C01819=1024.625,112.284,392.531,168.036,48.141,158.964
C01820=1024.630,112.533,392.511,168.039,48.136,158.963
C01821=1024.636,112.782,392.492,168.042,48.132,158.963
C01822=1024.642,113.032,392.473,168.044,48.128,158.962
C01823=1024.648,113.281,392.453,168.047,48.124,158.962
C01824=1024.654,113.530,392.434,168.049,48.119,158.962
C01825=1024.659,113.780,392.414,168.052,48.115,158.961
C01826=1024.665,114.028,392.395,168.055,48.111,158.961
C01827=1024.670,114.277,392.376,168.057,48.107,158.960
C01828=1024.676,114.527,392.356,168.060,48.103,158.960
C01829=1024.681,114.776,392.336,168.063,48.099,158.959
C01830=1024.687,115.025,392.317,168.065,48.094,158.959
C01831=1024.693,115.274,392.297,168.069,48.090,158.959
C01832=1024.699,115.523,392.277,168.072,48.086,158.958
C01833=1024.704,115.773,392.258,168.074,48.082,158.958
C01834=1024.710,116.022,392.238,168.077,48.077,158.957
C01835=1024.716,116.271,392.219,168.080,48.073,158.957
C01836=1024.722,116.520,392.199,168.082,48.069,158.956
C01837=1024.727,116.770,392.179,168.085,48.065,158.956
C01838=1024.733,117.018,392.159,168.087,48.061,158.955
C01839=1024.738,117.267,392.140,168.090,48.057,158.955
C01840=1024.744,117.517,392.121,168.094,48.052,158.955
C01841=1024.750,117.765,392.101,168.097,48.048,158.954
C01842=1024.755,118.015,392.082,168.099,48.044,158.954
C01843=1024.761,118.264,392.062,168.102,48.040,158.953
C01844=1024.766,118.513,392.042,168.104,48.035,158.953
C01845=1024.772,118.762,392.022,168.107,48.031,158.952
C01846=1024.778,119.012,392.003,168.110,48.027,158.952
C01847=1024.784,119.260,391.983,168.112,48.022,158.951
C01848=1024.790,119.510,391.964,168.116,48.018,158.951
C01849=1024.796,119.759,391.944,168.118,48.014,158.950
C01850=1024.801,120.008,391.924,168.121,48.010,158.950
C01851=1024.807,120.257,391.904,168.124,48.005,158.950
C01852=1024.812,120.507,391.885,168.127,48.002,158.949
C01853=1024.818,120.755,391.865,168.129,47.997,158.949
C01854=1024.824,121.005,391.845,168.132,47.993,158.948
C01855=1024.830,121.254,391.826,168.135,47.988,158.948
C01856=1024.836,121.502,391.806,168.138,47.984,158.947
C01857=1024.842,121.752,391.786,168.141,47.980,158.947
C01858=1024.847,122.001,391.766,168.143,47.976,158.946
C01859=1024.853,122.250,391.747,168.146,47.972,158.946
C01860=1024.859,122.500,391.726,168.149,47.967,158.946
C01861=1024.865,122.749,391.706,168.152,47.963,158.945
C01862=1024.871,122.998,391.687,168.155,47.959,158.945
C01863=1024.877,123.247,391.667,168.157,47.954,158.944
C01864=1024.883,123.531,391.644,168.161,47.949,158.944
C01865=1024.890,123.815,391.621,168.164,47.945,158.943
C01866=1024.896,124.099,391.599,168.167,47.940,158.943
C01867=1024.903,124.383,391.577,168.170,47.935,158.942
C01868=1024.909,124.632,391.558,168.173,47.931,158.942
C01869=1024.914,124.882,391.537,168.176,47.926,158.941
C01870=1024.920,125.131,391.517,168.179,47.922,158.941
C01871=1024.926,125.380,391.497,168.182,47.918,158.940
C01872=1024.932,125.629,391.477,168.184,47.913,158.940
C01873=1024.938,125.878,391.457,168.187,47.909,158.939
C01874=1024.944,126.127,391.438,168.191,47.905,158.939
C01875=1024.949,126.376,391.418,168.193,47.901,158.938
C01876=1024.955,126.625,391.398,168.196,47.896,158.938
C01877=1024.961,126.874,391.378,168.198,47.892,158.937
C01878=1024.967,127.124,391.358,168.202,47.888,158.937
C01879=1024.973,127.373,391.338,168.205,47.883,158.937
C01880=1024.979,127.622,391.318,168.207,47.879,158.936
C01881=1024.984,127.872,391.298,168.210,47.875,158.936
C01882=1024.990,128.120,391.278,168.214,47.870,158.935
C01883=1024.996,128.369,391.258,168.216,47.866,158.935
C01884=1025.003,128.619,391.238,168.219,47.862,158.934
C01885=1025.009,128.868,391.219,168.221,47.857,158.934
C01886=1025.015,129.117,391.199,168.225,47.853,158.933
C01887=1025.020,129.366,391.178,168.228,47.849,158.933
C01888=1025.026,129.615,391.158,168.230,47.844,158.932
C01889=1025.032,129.864,391.138,168.233,47.841,158.932
C01890=1025.038,130.114,391.119,168.237,47.836,158.932
C01891=1025.043,130.363,391.098,168.239,47.832,158.931
C01892=1025.049,130.612,391.078,168.242,47.828,158.931
C01893=1025.055,130.861,391.058,168.245,47.824,158.930
C01894=1025.061,131.110,391.038,168.247,47.819,158.930
C01895=1025.066,131.359,391.017,168.251,47.815,158.929
C01896=1025.072,131.608,390.997,168.254,47.811,158.929
C01897=1025.078,131.857,390.976,168.256,47.807,158.928
C01898=1025.084,132.106,390.956,168.259,47.802,158.928
C01899=1025.089,132.355,390.936,168.262,47.799,158.928
C01900=1025.095,132.604,390.916,168.265,47.794,158.927
C01901=1025.101,132.854,390.895,168.268,47.790,158.927
C01902=1025.107,133.103,390.875,168.271,47.786,158.926
C01903=1025.112,133.352,390.855,168.273,47.782,158.926
C01904=1025.118,133.601,390.835,168.276,47.777,158.925
C01905=1025.123,133.850,390.814,168.280,47.773,158.925
C01906=1025.130,134.099,390.794,168.282,47.769,158.924
C01907=1025.135,134.349,390.773,168.285,47.765,158.924
C01908=1025.141,134.597,390.753,168.288,47.761,158.924
C01909=1025.146,134.846,390.733,168.291,47.756,158.923
C01910=1025.153,135.095,390.712,168.294,47.753,158.923
C01911=1025.159,135.344,390.691,168.297,47.748,158.922
C01912=1025.165,135.593,390.671,168.300,47.744,158.922
C01913=1025.170,135.842,390.650,168.303,47.740,158.921
C01914=1025.176,136.092,390.630,168.306,47.736,158.921
C01915=1025.182,136.341,390.610,168.309,47.731,158.921
C01916=1025.187,136.590,390.589,168.311,47.727,158.920
C01917=1025.193,136.839,390.569,168.314,47.723,158.920
C01918=1025.199,137.088,390.547,168.318,47.719,158.919
C01919=1025.205,137.337,390.528,168.320,47.714,158.919
C01920=1025.210,137.586,390.507,168.323,47.711,158.918
C01921=1025.216,137.836,390.486,168.326,47.706,158.918
C01922=1025.222,138.085,390.466,168.329,47.702,158.918
C01923=1025.228,138.333,390.445,168.332,47.698,158.917
C01924=1025.234,138.582,390.425,168.335,47.694,158.917
C01925=1025.240,138.832,390.404,168.338,47.690,158.916
C01926=1025.245,139.081,390.383,168.341,47.685,158.916
C01927=1025.250,139.330,390.362,168.344,47.682,158.915
C01928=1025.257,139.614,390.339,168.348,47.677,158.915
C01929=1025.264,139.898,390.315,168.351,47.672,158.915
C01930=1025.270,140.182,390.291,168.354,47.668,158.914
C01931=1025.277,140.465,390.268,168.357,47.663,158.914
C01932=1025.282,140.714,390.247,168.361,47.658,158.913
C01933=1025.288,140.964,390.226,168.364,47.654,158.913
C01934=1025.294,141.213,390.205,168.366,47.651,158.912
C01935=1025.299,141.462,390.184,168.369,47.646,158.912
C01936=1025.306,141.711,390.164,168.373,47.642,158.911
C01937=1025.311,141.960,390.143,168.375,47.638,158.911
C01938=1025.316,142.209,390.122,168.378,47.634,158.911
C01939=1025.323,142.458,390.101,168.381,47.630,158.910
C01940=1025.329,142.707,390.081,168.384,47.625,158.910
C01941=1025.334,142.956,390.060,168.387,47.622,158.909
C01942=1025.340,143.205,390.039,168.390,47.617,158.909
C01943=1025.345,143.455,390.018,168.393,47.613,158.908
C01944=1025.351,143.703,389.997,168.397,47.609,158.908
C01945=1025.357,143.953,389.976,168.399,47.605,158.908
C01946=1025.363,144.201,389.955,168.402,47.601,158.907
C01947=1025.369,144.451,389.934,168.405,47.596,158.907
C01948=1025.374,144.700,389.914,168.408,47.592,158.906
C01949=1025.380,144.949,389.892,168.411,47.589,158.906
C01950=1025.386,145.198,389.872,168.415,47.584,158.905
C01951=1025.392,145.447,389.851,168.418,47.580,158.905
C01952=1025.398,145.696,389.830,168.420,47.576,158.905
C01953=1025.403,145.945,389.809,168.423,47.572,158.904
C01954=1025.409,146.195,389.788,168.427,47.568,158.904
C01955=1025.415,146.443,389.766,168.429,47.563,158.903
C01956=1025.420,146.692,389.745,168.432,47.560,158.903
C01957=1025.426,146.942,389.724,168.436,47.556,158.903
C01958=1025.432,147.190,389.703,168.439,47.551,158.902
C01959=1025.438,147.440,389.683,168.441,47.547,158.902
C01960=1025.444,147.688,389.661,168.445,47.543,158.901
C01961=1025.450,147.937,389.640,168.448,47.539,158.901
C01962=1025.454,148.187,389.619,168.451,47.535,158.900
C01963=1025.460,148.435,389.597,168.453,47.531,158.900
C01964=1025.466,148.684,389.576,168.457,47.527,158.900
C01965=1025.471,148.934,389.555,168.460,47.523,158.899
C01966=1025.478,149.183,389.533,168.463,47.519,158.899
C01967=1025.483,149.431,389.512,168.466,47.514,158.898
C01968=1025.489,149.681,389.491,168.469,47.511,158.898
C01969=1025.495,149.930,389.470,168.472,47.507,158.898
C01970=1025.501,150.179,389.448,168.476,47.502,158.897
C01971=1025.506,150.428,389.428,168.478,47.498,158.897
C01972=1025.512,150.677,389.406,168.481,47.495,158.896
C01973=1025.518,150.926,389.385,168.485,47.491,158.896
C01974=1025.524,151.175,389.363,168.488,47.486,158.896
C01975=1025.529,151.424,389.343,168.490,47.482,158.895
C01976=1025.535,151.673,389.321,168.494,47.478,158.895
C01977=1025.541,151.922,389.300,168.497,47.474,158.894
C01978=1025.547,152.171,389.278,168.500,47.470,158.894
C01979=1025.553,152.419,389.257,168.504,47.466,158.894
C01980=1025.558,152.669,389.235,168.506,47.462,158.893
C01981=1025.563,152.918,389.214,168.509,47.458,158.893
C01982=1025.569,153.167,389.193,168.513,47.454,158.892
C01983=1025.575,153.416,389.171,168.516,47.450,158.892
C01984=1025.581,153.665,389.150,168.518,47.446,158.892
C01985=1025.587,153.913,389.128,168.522,47.442,158.891
C01986=1025.593,154.163,389.107,168.525,47.438,158.891
C01987=1025.598,154.413,389.085,168.528,47.434,158.890
C01988=1025.604,154.661,389.064,168.531,47.429,158.890
C01989=1025.610,154.910,389.042,168.534,47.426,158.890
C01990=1025.615,155.159,389.021,168.537,47.422,158.889
C01991=1025.621,155.408,388.999,168.541,47.418,158.889
C01992=1025.628,155.692,388.974,168.544,47.413,158.888
C01993=1025.634,155.975,388.950,168.548,47.409,158.888
C01994=1025.640,156.259,388.925,168.552,47.404,158.887
C01995=1025.647,156.542,388.900,168.555,47.399,158.887
C01996=1025.653,156.792,388.879,168.558,47.395,158.887
C01997=1025.659,157.040,388.857,168.561,47.392,158.886
C01998=1025.664,157.290,388.835,168.565,47.388,158.886
C01999=1025.670,157.538,388.814,168.568,47.384,158.886
C02000=1025.676,157.787,388.792,168.570,47.379,158.885
C02001=1025.682,158.037,388.771,168.574,47.375,158.885
C02002=1025.687,158.285,388.749,168.577,47.372,158.884
C02003=1025.693,158.535,388.727,168.581,47.368,158.884
C02004=1025.699,158.783,388.706,168.583,47.363,158.883
C02005=1025.705,159.032,388.684,168.586,47.359,158.883
C02006=1025.711,159.281,388.663,168.590,47.355,158.883
C02007=1025.716,159.530,388.641,168.593,47.352,158.882
C02008=1025.721,159.771,388.619,168.596,47.348,158.882
C02009=1025.727,160.013,388.598,168.599,47.344,158.882
C02010=1025.732,160.254,388.576,168.602,47.340,158.881
C02011=1025.737,160.495,388.555,168.605,47.336,158.881
C02012=1025.743,160.737,388.534,168.608,47.333,158.881
C02013=1025.748,160.978,388.512,168.611,47.330,158.880
C02014=1025.753,161.220,388.491,168.614,47.326,158.880
C02015=1025.758,161.460,388.469,168.618,47.322,158.880
C02016=1025.765,161.709,388.447,168.621,47.318,158.879
C02017=1025.770,161.958,388.425,168.624,47.314,158.879
C02018=1025.775,162.207,388.403,168.628,47.310,158.879
C02019=1025.781,162.457,388.380,168.631,47.307,158.878
C02020=1025.787,162.705,388.358,168.633,47.303,158.878
C02021=1025.792,162.954,388.336,168.637,47.299,158.878
C02022=1025.798,163.203,388.313,168.640,47.295,158.877
C02023=1025.804,163.452,388.292,168.643,47.291,158.877
C02024=1025.809,163.701,388.270,168.647,47.287,158.876
C02025=1025.814,163.950,388.247,168.650,47.284,158.876
C02026=1025.820,164.199,388.225,168.654,47.280,158.876
C02027=1025.826,164.447,388.203,168.656,47.276,158.875
C02028=1025.831,164.697,388.180,168.659,47.272,158.875
C02029=1025.837,164.946,388.159,168.663,47.268,158.875
C02030=1025.842,165.194,388.136,168.666,47.264,158.874
C02031=1025.848,165.444,388.114,168.669,47.261,158.874
C02032=1025.854,165.692,388.092,168.673,47.257,158.874
C02033=1025.860,165.942,388.069,168.676,47.253,158.873
C02034=1025.865,166.190,388.047,168.680,47.249,158.873
C02035=1025.870,166.439,388.025,168.682,47.245,158.873
C02036=1025.877,166.688,388.002,168.685,47.241,158.872
C02037=1025.882,166.938,387.980,168.689,47.237,158.872
C02038=1025.887,167.186,387.957,168.692,47.234,158.871
C02039=1025.893,167.435,387.936,168.696,47.230,158.871
C02040=1025.899,167.684,387.913,168.699,47.226,158.871
C02041=1025.905,167.933,387.891,168.703,47.222,158.870
C02042=1025.910,168.181,387.869,168.706,47.218,158.870
C02043=1025.916,168.431,387.846,168.708,47.215,158.870
C02044=1025.922,168.680,387.823,168.712,47.211,158.869
C02045=1025.927,168.929,387.801,168.715,47.207,158.869
C02046=1025.933,169.178,387.779,168.719,47.203,158.869
C02047=1025.939,169.426,387.756,168.722,47.199,158.868
C02048=1025.944,169.675,387.734,168.726,47.195,158.868
C02049=1025.951,169.924,387.712,168.729,47.191,158.868
C02050=1025.956,170.174,387.689,168.733,47.187,158.867
C02051=1025.962,170.422,387.667,168.735,47.184,158.867
C02052=1025.967,170.671,387.644,168.739,47.180,158.867
C02053=1025.973,170.920,387.622,168.742,47.176,158.866
C02054=1025.979,171.169,387.599,168.746,47.172,158.866
C02055=1025.984,171.418,387.576,168.749,47.168,158.865
C02056=1025.992,171.717,387.549,168.752,47.164,158.865
C02057=1025.998,172.015,387.523,168.757,47.159,158.865
C02058=1026.005,172.314,387.495,168.761,47.154,158.864
C02059=1026.012,172.613,387.468,168.766,47.150,158.864
C02060=1026.017,172.862,387.446,168.768,47.146,158.863
C02061=1026.024,173.110,387.424,168.772,47.142,158.863
C02062=1026.029,173.359,387.401,168.775,47.138,158.863
C02063=1026.035,173.608,387.378,168.779,47.134,158.862
C02064=1026.041,173.857,387.357,168.782,47.131,158.862
C02065=1026.047,174.106,387.334,168.786,47.127,158.862
C02066=1026.053,174.355,387.311,168.789,47.123,158.861
C02067=1026.058,174.604,387.288,168.793,47.119,158.861
C02068=1026.065,174.853,387.266,168.795,47.115,158.861
C02069=1026.070,175.102,387.243,168.799,47.111,158.860
C02070=1026.076,175.351,387.220,168.803,47.107,158.860
C02071=1026.082,175.600,387.197,168.806,47.104,158.860
C02072=1026.088,175.848,387.175,168.810,47.100,158.859
C02073=1026.094,176.098,387.153,168.813,47.096,158.859
C02074=1026.099,176.347,387.130,168.817,47.092,158.859
C02075=1026.105,176.595,387.107,168.820,47.088,158.858
C02076=1026.111,176.844,387.085,168.824,47.084,158.858
C02077=1026.117,177.092,387.062,168.827,47.080,158.858
C02078=1026.122,177.341,387.039,168.830,47.076,158.857
C02079=1026.128,177.590,387.016,168.834,47.072,158.857
C02080=1026.135,177.839,386.994,168.837,47.069,158.856
C02081=1026.141,178.089,386.971,168.841,47.065,158.856
C02082=1026.146,178.338,386.948,168.845,47.061,158.856
C02083=1026.152,178.587,386.925,168.848,47.057,158.855
C02084=1026.159,178.835,386.903,168.852,47.053,158.855
C02085=1026.164,179.084,386.880,168.855,47.049,158.855
C02086=1026.170,179.333,386.857,168.858,47.045,158.854
C02087=1026.176,179.582,386.834,168.862,47.041,158.854
C02088=1026.182,179.831,386.812,168.865,47.038,158.854
C02089=1026.188,180.080,386.789,168.869,47.034,158.853
C02090=1026.194,180.328,386.766,168.873,47.030,158.853
C02091=1026.200,180.577,386.743,168.876,47.026,158.853
C02092=1026.206,180.826,386.720,168.880,47.022,158.852
C02093=1026.212,181.075,386.697,168.883,47.018,158.852
C02094=1026.217,181.324,386.674,168.887,47.015,158.852
C02095=1026.223,181.573,386.652,168.890,47.011,158.851
C02096=1026.230,181.822,386.629,168.893,47.007,158.851
C02097=1026.236,182.071,386.606,168.897,47.003,158.851
C02098=1026.242,182.320,386.583,168.901,47.000,158.850
C02099=1026.247,182.569,386.560,168.904,46.996,158.850
C02100=1026.253,182.818,386.537,168.908,46.992,158.850
C02101=1026.259,183.066,386.513,168.912,46.988,158.849
C02102=1026.264,183.315,386.490,168.915,46.985,158.849
C02103=1026.270,183.564,386.467,168.919,46.981,158.849
C02104=1026.276,183.813,386.442,168.922,46.977,158.849
C02105=1026.282,184.062,386.419,168.926,46.974,158.848
C02106=1026.287,184.311,386.396,168.929,46.970,158.848
C02107=1026.293,184.560,386.372,168.933,46.967,158.848
C02108=1026.298,184.808,386.349,168.936,46.963,158.847
C02109=1026.304,185.057,386.326,168.940,46.959,158.847
C02110=1026.309,185.306,386.302,168.944,46.956,158.847
C02111=1026.315,185.555,386.279,168.947,46.952,158.847
C02112=1026.320,185.803,386.255,168.951,46.948,158.846
C02113=1026.326,186.052,386.232,168.954,46.945,158.846
C02114=1026.332,186.301,386.208,168.958,46.941,158.846
C02115=1026.338,186.551,386.184,168.962,46.938,158.846
C02116=1026.343,186.799,386.161,168.965,46.934,158.845
C02117=1026.349,187.048,386.138,168.969,46.930,158.845
C02118=1026.354,187.297,386.114,168.972,46.927,158.845
C02119=1026.361,187.545,386.090,168.976,46.923,158.844
C02120=1026.367,187.828,386.063,168.980,46.919,158.844
C02121=1026.373,188.111,386.037,168.984,46.916,158.844
C02122=1026.379,188.394,386.010,168.989,46.911,158.843
C02123=1026.386,188.676,385.983,168.993,46.907,158.843
C02124=1026.392,188.925,385.959,168.997,46.903,158.843
C02125=1026.397,189.174,385.936,169.000,46.900,158.843
C02126=1026.404,189.423,385.912,169.004,46.896,158.842
C02127=1026.409,189.672,385.888,169.008,46.893,158.842
C02128=1026.415,189.920,385.865,169.011,46.889,158.842
C02129=1026.421,190.169,385.842,169.015,46.886,158.841
C02130=1026.426,190.418,385.817,169.019,46.882,158.841
C02131=1026.433,190.667,385.793,169.022,46.879,158.841
C02132=1026.438,190.916,385.770,169.026,46.875,158.841
C02133=1026.444,191.164,385.746,169.030,46.871,158.840
C02134=1026.450,191.413,385.722,169.033,46.868,158.840
C02135=1026.455,191.662,385.699,169.037,46.864,158.840
C02136=1026.461,191.911,385.675,169.041,46.860,158.839
C02137=1026.467,192.159,385.651,169.044,46.857,158.839
C02138=1026.473,192.409,385.627,169.048,46.853,158.839
C02139=1026.479,192.657,385.604,169.052,46.850,158.839
C02140=1026.484,192.906,385.579,169.056,46.846,158.838
C02141=1026.490,193.155,385.556,169.059,46.843,158.838
C02142=1026.496,193.404,385.532,169.063,46.839,158.838
C02143=1026.502,193.652,385.508,169.067,46.835,158.837
C02144=1026.508,193.900,385.485,169.070,46.832,158.837
C02145=1026.514,194.150,385.461,169.074,46.828,158.837
C02146=1026.520,194.399,385.437,169.078,46.825,158.837
C02147=1026.525,194.647,385.413,169.082,46.821,158.836
C02148=1026.532,194.896,385.389,169.086,46.818,158.836
C02149=1026.537,195.145,385.364,169.089,46.814,158.836
C02150=1026.543,195.394,385.341,169.094,46.811,158.836
C02151=1026.549,195.643,385.317,169.098,46.807,158.835
C02152=1026.555,195.891,385.293,169.101,46.804,158.835
C02153=1026.561,196.140,385.269,169.105,46.800,158.835
C02154=1026.567,196.389,385.245,169.109,46.797,158.835
C02155=1026.573,196.637,385.221,169.113,46.793,158.834
C02156=1026.578,196.887,385.197,169.117,46.790,158.834
C02157=1026.584,197.135,385.174,169.120,46.786,158.834
C02158=1026.591,197.384,385.150,169.124,46.782,158.833
C02159=1026.596,197.633,385.125,169.128,46.779,158.833
C02160=1026.603,197.882,385.101,169.132,46.775,158.833
C02161=1026.608,198.130,385.077,169.136,46.772,158.833
C02162=1026.614,198.379,385.053,169.139,46.768,158.832
C02163=1026.620,198.628,385.029,169.143,46.765,158.832
C02164=1026.626,198.876,385.005,169.147,46.761,158.832
C02165=1026.632,199.126,384.981,169.151,46.757,158.832
C02166=1026.638,199.374,384.957,169.155,46.754,158.832
C02167=1026.645,199.623,384.933,169.159,46.750,158.831
C02168=1026.650,199.871,384.909,169.163,46.747,158.831
C02169=1026.657,200.120,384.885,169.166,46.743,158.831
C02170=1026.662,200.369,384.860,169.171,46.740,158.831
C02171=1026.668,200.618,384.836,169.175,46.737,158.830
C02172=1026.673,200.867,384.811,169.179,46.733,158.830
C02173=1026.679,201.116,384.787,169.182,46.730,158.830
C02174=1026.685,201.364,384.762,169.186,46.727,158.830
C02175=1026.691,201.613,384.738,169.190,46.723,158.829
C02176=1026.697,201.862,384.714,169.194,46.719,158.829
C02177=1026.702,202.111,384.689,169.197,46.716,158.829
C02178=1026.708,202.360,384.665,169.202,46.713,158.829
C02179=1026.715,202.608,384.640,169.206,46.709,158.828
C02180=1026.720,202.857,384.616,169.210,46.706,158.828
C02181=1026.726,203.106,384.591,169.214,46.703,158.828
C02182=1026.731,203.354,384.566,169.218,46.699,158.828
C02183=1026.737,203.603,384.541,169.221,46.696,158.828
C02184=1026.762,204.642,384.439,169.608,46.799,158.896
C02185=1026.772,205.034,384.399,169.613,46.795,158.896
C02186=1026.783,205.426,384.358,169.617,46.791,158.896
C02187=1026.794,205.817,384.317,169.622,46.786,158.895
C02188=1026.804,206.209,384.275,169.627,46.782,158.895
C02189=1026.810,206.457,384.249,169.629,46.780,158.895
C02190=1026.817,206.706,384.223,169.632,46.777,158.895
C02191=1026.824,206.954,384.197,169.636,46.775,158.895
C02192=1026.831,207.203,384.171,169.638,46.772,158.894
C02193=1026.837,207.451,384.145,169.641,46.770,158.894
C02194=1026.843,207.700,384.120,169.644,46.767,158.894
C02195=1026.850,207.949,384.093,169.647,46.765,158.894
C02196=1026.856,208.197,384.066,169.650,46.762,158.894
C02197=1026.863,208.445,384.040,169.654,46.759,158.893
C02198=1026.870,208.694,384.014,169.656,46.757,158.893
C02199=1026.877,208.943,383.988,169.659,46.754,158.893
C02200=1026.883,209.191,383.962,169.662,46.752,158.893
C02201=1026.890,209.440,383.935,169.665,46.749,158.893
C02202=1026.896,209.688,383.909,169.668,46.747,158.893
C02203=1026.903,209.937,383.883,169.671,46.745,158.892
C02204=1026.909,210.185,383.856,169.674,46.742,158.892
C02205=1026.916,210.434,383.830,169.677,46.739,158.892
C02206=1026.923,210.682,383.804,169.680,46.737,158.892
C02207=1026.930,210.931,383.777,169.683,46.734,158.892
C02208=1026.936,211.179,383.751,169.686,46.732,158.892
C02209=1026.942,211.427,383.725,169.689,46.730,158.892
C02210=1026.948,211.676,383.697,169.692,46.728,158.891
C02211=1026.955,211.924,383.671,169.695,46.725,158.891
C02212=1026.962,212.173,383.645,169.698,46.722,158.891
C02213=1026.968,212.421,383.618,169.701,46.720,158.891
C02214=1026.975,212.670,383.592,169.704,46.718,158.891
C02215=1026.981,212.919,383.565,169.707,46.715,158.891
C02216=1026.988,213.167,383.539,169.711,46.713,158.891
C02217=1026.994,213.416,383.512,169.713,46.711,158.890
C02218=1027.001,213.664,383.486,169.716,46.708,158.890
C02219=1027.008,213.913,383.459,169.720,46.706,158.890
C02220=1027.014,214.161,383.433,169.722,46.703,158.890
C02221=1027.021,214.410,383.406,169.726,46.701,158.890
C02222=1027.027,214.659,383.380,169.729,46.699,158.890
C02223=1027.034,214.907,383.353,169.731,46.696,158.890
C02224=1027.040,215.155,383.327,169.735,46.693,158.889
C02225=1027.047,215.404,383.299,169.737,46.691,158.889
C02226=1027.054,215.653,383.273,169.741,46.689,158.889
C02227=1027.060,215.901,383.246,169.744,46.687,158.889
C02228=1027.067,216.150,383.220,169.746,46.685,158.889
C02229=1027.073,216.398,383.193,169.750,46.682,158.889
C02230=1027.080,216.647,383.167,169.753,46.679,158.889
C02231=1027.087,216.895,383.140,169.756,46.677,158.888
C02232=1027.093,217.143,383.113,169.759,46.675,158.888
C02233=1027.100,217.392,383.087,169.762,46.673,158.888
C02234=1027.106,217.640,383.060,169.765,46.670,158.888
C02235=1027.113,217.889,383.034,169.768,46.668,158.888
C02236=1027.120,218.138,383.006,169.772,46.665,158.888
C02237=1027.126,218.386,382.980,169.775,46.663,158.888
C02238=1027.133,218.634,382.953,169.778,46.661,158.888
C02239=1027.140,218.883,382.926,169.781,46.658,158.887
C02240=1027.146,219.131,382.900,169.784,46.656,158.887
C02241=1027.157,219.527,382.857,169.789,46.653,158.887
C02242=1027.167,219.922,382.814,169.794,46.649,158.887
C02243=1027.177,220.318,382.770,169.799,46.645,158.887
C02244=1027.187,220.713,382.727,169.804,46.642,158.887
C02245=1027.194,220.962,382.701,169.806,46.640,158.887
C02246=1027.201,221.211,382.674,169.810,46.637,158.886
C02247=1027.207,221.459,382.646,169.813,46.635,158.886
C02248=1027.213,221.708,382.619,169.816,46.633,158.886
C02249=1027.221,221.956,382.592,169.819,46.631,158.886
C02250=1027.226,222.204,382.566,169.823,46.628,158.886
C02251=1027.233,222.453,382.538,169.825,46.626,158.886
C02252=1027.240,222.702,382.511,169.829,46.624,158.886
C02253=1027.246,222.949,382.484,169.832,46.622,158.886
C02254=1027.253,223.198,382.457,169.835,46.620,158.886
C02255=1027.259,223.447,382.429,169.838,46.618,158.886
C02256=1027.266,223.695,382.403,169.842,46.615,158.886
C02257=1027.273,223.943,382.376,169.844,46.613,158.885
C02258=1027.279,224.192,382.349,169.848,46.611,158.885
C02259=1027.286,224.440,382.321,169.851,46.609,158.885
C02260=1027.292,224.689,382.295,169.854,46.607,158.885
C02261=1027.299,224.937,382.267,169.857,46.604,158.885
C02262=1027.305,225.186,382.239,169.861,46.602,158.885
C02263=1027.313,225.434,382.213,169.864,46.600,158.885
C02264=1027.319,225.682,382.186,169.866,46.598,158.885
C02265=1027.325,225.931,382.159,169.870,46.595,158.885
C02266=1027.332,226.180,382.131,169.874,46.594,158.885
C02267=1027.339,226.428,382.104,169.876,46.591,158.885
C02268=1027.346,226.677,382.077,169.880,46.589,158.885
C02269=1027.352,226.925,382.049,169.883,46.587,158.884
C02270=1027.359,227.173,382.022,169.886,46.585,158.884
C02271=1027.365,227.422,381.995,169.889,46.582,158.884
C02272=1027.372,227.670,381.967,169.892,46.580,158.884
C02273=1027.379,227.919,381.940,169.895,46.579,158.884
C02274=1027.385,228.167,381.913,169.899,46.576,158.884
C02275=1027.391,228.415,381.885,169.902,46.574,158.884
C02276=1027.398,228.664,381.858,169.906,46.572,158.884
C02277=1027.405,228.912,381.830,169.908,46.570,158.884
C02278=1027.411,229.161,381.802,169.912,46.568,158.884
C02279=1027.417,229.409,381.775,169.915,46.566,158.884
C02280=1027.424,229.658,381.748,169.918,46.564,158.884
C02281=1027.430,229.906,381.720,169.922,46.562,158.884
C02282=1027.437,230.154,381.692,169.925,46.560,158.884
C02283=1027.444,230.403,381.665,169.927,46.558,158.883
C02284=1027.450,230.651,381.637,169.931,46.556,158.884
C02285=1027.457,230.899,381.609,169.935,46.554,158.883
C02286=1027.463,231.148,381.582,169.937,46.551,158.883
C02287=1027.470,231.396,381.554,169.941,46.550,158.883
C02288=1027.476,231.645,381.527,169.944,46.547,158.883
C02289=1027.483,231.894,381.499,169.947,46.545,158.883
C02290=1027.490,232.142,381.471,169.951,46.544,158.883
C02291=1027.496,232.390,381.444,169.954,46.541,158.883
C02292=1027.502,232.638,381.416,169.957,46.540,158.883
C02293=1027.508,232.887,381.388,169.960,46.538,158.883
C02294=1027.515,233.135,381.360,169.964,46.535,158.883
C02295=1027.522,233.384,381.333,169.967,46.534,158.883
C02296=1027.529,233.632,381.304,169.970,46.532,158.883
C02297=1027.538,234.020,381.261,169.975,46.529,158.883
C02298=1027.548,234.408,381.218,169.981,46.525,158.883
C02299=1027.559,234.795,381.175,169.986,46.522,158.883
C02300=1027.569,235.183,381.131,169.990,46.519,158.883
C02301=1027.576,235.431,381.103,169.994,46.518,158.883
C02302=1027.583,235.680,381.075,169.998,46.515,158.883
C02303=1027.589,235.928,381.048,170.001,46.514,158.883
C02304=1027.595,236.177,381.019,170.004,46.512,158.883
C02305=1027.602,236.425,380.991,170.008,46.510,158.883
C02306=1027.609,236.673,380.963,170.011,46.508,158.883
C02307=1027.616,236.922,380.935,170.014,46.506,158.883
C02308=1027.622,237.170,380.908,170.017,46.504,158.883
C02309=1027.629,237.419,380.880,170.021,46.502,158.883
C02310=1027.635,237.667,380.851,170.024,46.500,158.883
C02311=1027.642,237.915,380.823,170.027,46.498,158.883
C02312=1027.648,238.164,380.795,170.031,46.496,158.882
C02313=1027.655,238.412,380.768,170.034,46.494,158.883
C02314=1027.661,238.661,380.739,170.038,46.492,158.882
C02315=1027.668,238.909,380.711,170.041,46.491,158.883
C02316=1027.675,239.157,380.683,170.044,46.488,158.882
C02317=1027.681,239.406,380.656,170.048,46.487,158.882
C02318=1027.688,239.653,380.627,170.052,46.485,158.883
C02319=1027.694,239.902,380.599,170.054,46.483,158.882
C02320=1027.701,240.151,380.571,170.058,46.481,158.883
C02321=1027.708,240.398,380.543,170.061,46.479,158.882
C02322=1027.714,240.647,380.514,170.064,46.478,158.882
C02323=1027.721,240.895,380.486,170.068,46.476,158.883
C02324=1027.727,241.144,380.457,170.071,46.474,158.882
C02325=1027.734,241.391,380.429,170.075,46.472,158.883
C02326=1027.740,241.640,380.401,170.078,46.471,158.883
C02327=1027.747,241.888,380.372,170.082,46.469,158.883
C02328=1027.753,242.137,380.344,170.085,46.467,158.883
C02329=1027.760,242.385,380.315,170.088,46.465,158.883
C02330=1027.766,242.633,380.287,170.091,46.463,158.883
C02331=1027.773,242.881,380.259,170.095,46.461,158.883
C02332=1027.779,243.130,380.231,170.099,46.459,158.883
C02333=1027.786,243.378,380.202,170.101,46.458,158.883
C02334=1027.793,243.627,380.174,170.105,46.456,158.883
C02335=1027.799,243.875,380.145,170.109,46.454,158.883
C02336=1027.806,244.123,380.117,170.112,46.452,158.883
C02337=1027.812,244.372,380.088,170.115,46.451,158.883
C02338=1027.818,244.620,380.059,170.119,46.449,158.883
C02339=1027.824,244.869,380.031,170.123,46.448,158.883
C02340=1027.831,245.116,380.002,170.125,46.446,158.883
C02341=1027.838,245.364,379.973,170.129,46.445,158.883
C02342=1027.844,245.613,379.944,170.133,46.442,158.883
C02343=1027.850,245.861,379.916,170.136,46.441,158.883
C02344=1027.857,246.109,379.887,170.139,46.439,158.883
C02345=1027.863,246.357,379.858,170.143,46.438,158.883
C02346=1027.870,246.606,379.829,170.147,46.436,158.883
C02347=1027.877,246.855,379.801,170.149,46.434,158.883
C02348=1027.883,247.103,379.772,170.153,46.433,158.883
C02349=1027.889,247.351,379.743,170.157,46.431,158.883
C02350=1027.895,247.599,379.714,170.161,46.429,158.883
C02351=1027.902,247.847,379.686,170.163,46.428,158.883
C02352=1027.908,248.095,379.657,170.167,46.426,158.884
C02353=1027.918,248.477,379.612,170.173,46.424,158.884
C02354=1027.928,248.859,379.568,170.178,46.421,158.884
C02355=1027.938,249.241,379.524,170.183,46.419,158.884
C02356=1027.949,249.622,379.479,170.188,46.416,158.884
C02357=1027.955,249.870,379.450,170.192,46.414,158.884
C02358=1027.962,250.119,379.421,170.196,46.413,158.884
C02359=1027.968,250.368,379.392,170.200,46.411,158.884
C02360=1027.975,250.616,379.364,170.202,46.410,158.884
C02361=1027.981,250.864,379.335,170.206,46.408,158.884
C02362=1027.988,251.113,379.306,170.210,46.406,158.884
C02363=1027.994,251.361,379.277,170.214,46.405,158.884
C02364=1028.000,251.609,379.247,170.217,46.403,158.884
C02365=1028.007,251.857,379.219,170.220,46.402,158.884
C02366=1028.014,252.105,379.190,170.224,46.400,158.884
C02367=1028.020,252.354,379.161,170.228,46.398,158.885
C02368=1028.027,252.602,379.132,170.232,46.397,158.885
C02369=1028.034,252.850,379.103,170.235,46.396,158.885
C02370=1028.040,253.098,379.074,170.238,46.394,158.885
C02371=1028.047,253.346,379.045,170.242,46.393,158.885
C02372=1028.053,253.594,379.015,170.246,46.391,158.885
C02373=1028.061,253.843,378.986,170.250,46.389,158.885
C02374=1028.067,254.091,378.957,170.252,46.388,158.885
C02375=1028.073,254.339,378.928,170.256,46.386,158.885
C02376=1028.080,254.588,378.899,170.260,46.384,158.885
C02377=1028.086,254.836,378.870,170.264,46.383,158.885
C02378=1028.093,255.084,378.841,170.267,46.381,158.885
C02379=1028.100,255.332,378.812,170.270,46.380,158.885
C02380=1028.107,255.580,378.782,170.274,46.378,158.886
C02381=1028.113,255.828,378.753,170.278,46.377,158.886
C02382=1028.121,256.077,378.724,170.282,46.375,158.886
C02383=1028.127,256.325,378.695,170.285,46.374,158.886
C02384=1028.133,256.573,378.666,170.289,46.372,158.886
C02385=1028.140,256.821,378.636,170.293,46.370,158.886
C02386=1028.147,257.069,378.607,170.296,46.369,158.886
C02387=1028.154,257.318,378.578,170.299,46.367,158.886
C02388=1028.160,257.566,378.549,170.304,46.366,158.886
C02389=1028.168,257.814,378.519,170.307,46.365,158.887
C02390=1028.174,258.062,378.490,170.311,46.363,158.887
C02391=1028.180,258.310,378.461,170.315,46.361,158.887
C02392=1028.188,258.559,378.432,170.319,46.360,158.887
C02393=1028.194,258.806,378.402,170.321,46.358,158.887
C02394=1028.201,259.055,378.373,170.325,46.357,158.887
C02395=1028.207,259.303,378.344,170.329,46.356,158.887
C02396=1028.214,259.552,378.314,170.333,46.354,158.887
C02397=1028.221,259.799,378.285,170.337,46.352,158.887
C02398=1028.228,260.048,378.256,170.341,46.351,158.887
C02399=1028.235,260.296,378.226,170.344,46.350,158.888
C02400=1028.242,260.545,378.197,170.348,46.348,158.888
C02401=1028.248,260.792,378.167,170.351,46.347,158.888
C02402=1028.255,261.041,378.137,170.355,46.346,158.888
C02403=1028.262,261.288,378.108,170.359,46.344,158.888
C02404=1028.268,261.537,378.079,170.362,46.342,158.888
C02405=1028.275,261.785,378.049,170.366,46.341,158.888
C02406=1028.281,262.033,378.020,170.370,46.340,158.888
C02407=1028.288,262.281,377.989,170.373,46.339,158.889
C02408=1028.294,262.529,377.959,170.377,46.337,158.889
C02409=1028.305,262.909,377.914,170.383,46.335,158.889
C02410=1028.315,263.290,377.868,170.389,46.333,158.889
C02411=1028.325,263.670,377.822,170.395,46.331,158.889
C02412=1028.335,264.050,377.777,170.400,46.329,158.890
C02413=1028.342,264.299,377.747,170.404,46.327,158.890
C02414=1028.348,264.546,377.717,170.408,46.326,158.890
C02415=1028.356,264.794,377.687,170.412,46.325,158.890
C02416=1028.361,265.043,377.657,170.415,46.324,158.890
C02417=1028.368,265.291,377.627,170.419,46.322,158.890
C02418=1028.375,265.539,377.597,170.423,46.321,158.891
C02419=1028.382,265.787,377.567,170.427,46.320,158.891
C02420=1028.389,266.036,377.538,170.431,46.319,158.891
C02421=1028.395,266.283,377.507,170.434,46.317,158.891
C02422=1028.402,266.532,377.477,170.438,46.316,158.891
C02423=1028.408,266.779,377.448,170.442,46.315,158.891
C02424=1028.415,267.028,377.417,170.445,46.314,158.891
C02425=1028.421,267.275,377.387,170.449,46.313,158.892
C02426=1028.428,267.523,377.357,170.453,46.311,158.892
C02427=1028.435,267.772,377.326,170.457,46.310,158.892
C02428=1028.441,268.020,377.297,170.461,46.309,158.892
C02429=1028.448,268.268,377.267,170.465,46.307,158.892
C02430=1028.454,268.516,377.237,170.469,46.306,158.893
C02431=1028.461,268.764,377.207,170.473,46.305,158.893
C02432=1028.468,269.013,377.176,170.477,46.304,158.893
C02433=1028.474,269.260,377.146,170.480,46.303,158.893
C02434=1028.481,269.509,377.116,170.484,46.302,158.893
C02435=1028.488,269.757,377.085,170.488,46.300,158.893
C02436=1028.494,270.005,377.056,170.492,46.299,158.894
C02437=1028.502,270.252,377.025,170.496,46.298,158.894
C02438=1028.508,270.501,376.994,170.500,46.297,158.894
C02439=1028.515,270.748,376.964,170.503,46.295,158.894
C02440=1028.521,270.997,376.934,170.507,46.294,158.894
C02441=1028.528,271.245,376.903,170.511,46.293,158.895
C02442=1028.534,271.493,376.873,170.516,46.292,158.895
C02443=1028.541,271.741,376.842,170.519,46.292,158.895
C02444=1028.548,271.989,376.811,170.522,46.290,158.895
C02445=1028.554,272.237,376.781,170.526,46.289,158.895
C02446=1028.561,272.485,376.751,170.530,46.288,158.896
C02447=1028.567,272.733,376.720,170.534,46.287,158.896
C02448=1028.575,272.982,376.690,170.538,46.286,158.896
C02449=1028.581,273.229,376.659,170.543,46.285,158.896
C02450=1028.588,273.477,376.629,170.546,46.283,158.896
C02451=1028.594,273.726,376.598,170.550,46.282,158.897
C02452=1028.600,273.973,376.567,170.554,46.281,158.897
C02453=1028.608,274.221,376.537,170.558,46.280,158.897
C02454=1028.614,274.470,376.506,170.562,46.279,158.897
C02455=1028.621,274.717,376.476,170.566,46.278,158.898
C02456=1028.627,274.965,376.445,170.570,46.277,158.898
C02457=1028.634,275.213,376.414,170.574,46.276,158.898
C02458=1028.641,275.461,376.384,170.578,46.275,158.898
C02459=1028.648,275.710,376.353,170.582,46.274,158.899
C02460=1028.654,275.958,376.321,170.586,46.273,158.899
C02461=1028.661,276.205,376.292,170.590,46.272,158.899
C02462=1028.667,276.454,376.261,170.594,46.271,158.899
C02463=1028.675,276.701,376.230,170.598,46.270,158.900
C02464=1028.681,276.950,376.199,170.602,46.269,158.900
C02465=1028.692,277.335,376.152,170.608,46.268,158.900
C02466=1028.701,277.719,376.104,170.614,46.266,158.901
C02467=1028.712,278.104,376.056,170.621,46.264,158.901
C02468=1028.722,278.489,376.007,170.627,46.263,158.901
C02469=1028.729,278.737,375.976,170.631,46.262,158.902
C02470=1028.736,278.985,375.944,170.635,46.261,158.902
C02471=1028.742,279.233,375.915,170.639,46.260,158.902
C02472=1028.749,279.481,375.883,170.644,46.259,158.902
C02473=1028.756,279.728,375.852,170.647,46.259,158.903
C02474=1028.762,279.977,375.821,170.651,46.258,158.903
C02475=1028.769,280.225,375.790,170.655,46.257,158.903
C02476=1028.776,280.473,375.758,170.659,46.256,158.903
C02477=1028.782,280.721,375.727,170.663,46.255,158.904
C02478=1028.789,280.969,375.696,170.667,46.254,158.904
C02479=1028.796,281.217,375.665,170.671,46.253,158.904
C02480=1028.803,281.465,375.634,170.675,46.252,158.905
C02481=1028.809,281.712,375.603,170.679,46.251,158.905
C02482=1028.816,281.960,375.571,170.683,46.250,158.905
C02483=1028.822,282.208,375.541,170.688,46.250,158.905
C02484=1028.829,282.456,375.509,170.692,46.249,158.906
C02485=1028.836,282.704,375.478,170.696,46.248,158.906
C02486=1028.842,282.952,375.446,170.700,46.247,158.906
C02487=1028.849,283.200,375.415,170.704,46.246,158.907
C02488=1028.856,283.448,375.383,170.708,46.245,158.907
C02489=1028.863,283.695,375.353,170.712,46.244,158.907
C02490=1028.870,283.943,375.321,170.716,46.244,158.907
C02491=1028.877,284.191,375.290,170.720,46.243,158.908
C02492=1028.883,284.440,375.259,170.724,46.242,158.908
C02493=1028.890,284.688,375.228,170.730,46.241,158.908
C02494=1028.897,284.936,375.196,170.734,46.240,158.909
C02495=1028.903,285.183,375.165,170.738,46.239,158.909
C02496=1028.910,285.431,375.133,170.742,46.238,158.909
C02497=1028.917,285.679,375.102,170.746,46.238,158.910
C02498=1028.924,285.927,375.070,170.750,46.237,158.910
C02499=1028.931,286.174,375.038,170.755,46.237,158.910
C02500=1028.938,286.423,375.006,170.759,46.235,158.910
C02501=1028.945,286.671,374.975,170.763,46.234,158.911
C02502=1028.951,286.919,374.944,170.767,46.234,158.911
C02503=1028.958,287.167,374.912,170.771,46.233,158.911
C02504=1028.965,287.415,374.881,170.775,46.233,158.912
C02505=1028.972,287.662,374.849,170.779,46.232,158.912
C02506=1028.979,287.910,374.817,170.784,46.231,158.912
C02507=1028.985,288.158,374.785,170.788,46.230,158.913
C02508=1028.991,288.406,374.754,170.792,46.230,158.913
C02509=1028.998,288.653,374.722,170.796,46.229,158.913
C02510=1029.005,288.901,374.690,170.800,46.228,158.914
C02511=1029.012,289.149,374.659,170.805,46.228,158.914
C02512=1029.019,289.398,374.627,170.809,46.227,158.914
C02513=1029.025,289.645,374.594,170.814,46.226,158.915
C02514=1029.032,289.893,374.563,170.818,46.225,158.915
C02515=1029.039,290.140,374.531,170.823,46.225,158.915
C02516=1029.046,290.388,374.499,170.827,46.224,158.916
C02517=1029.053,290.636,374.468,170.831,46.224,158.916
C02518=1029.059,290.885,374.435,170.835,46.223,158.917
C02519=1029.066,291.132,374.403,170.839,46.222,158.917
C02520=1029.073,291.380,374.371,170.844,46.222,158.917
C02521=1029.084,291.777,374.320,170.851,46.221,158.918
C02522=1029.095,292.175,374.269,170.857,46.220,158.918
C02523=1029.106,292.571,374.218,170.865,46.219,158.919
C02524=1029.117,292.968,374.166,170.871,46.218,158.919
C02525=1029.123,293.216,374.134,170.875,46.217,158.920
C02526=1029.130,293.464,374.102,170.881,46.217,158.920
C02527=1029.138,293.712,374.070,170.885,46.216,158.921
C02528=1029.144,293.959,374.037,170.889,46.215,158.921
C02529=1029.151,294.207,374.005,170.893,46.215,158.921
C02530=1029.157,294.455,373.973,170.898,46.215,158.922
C02531=1029.165,294.703,373.940,170.902,46.214,158.922
C02532=1029.171,294.951,373.907,170.906,46.214,158.923
C02533=1029.177,295.199,373.875,170.911,46.213,158.923
C02534=1029.184,295.446,373.843,170.915,46.213,158.923
C02535=1029.190,295.694,373.811,170.919,46.213,158.924
C02536=1029.197,295.942,373.777,170.925,46.212,158.924
C02537=1029.204,296.189,373.745,170.929,46.212,158.925
C02538=1029.210,296.437,373.713,170.933,46.211,158.925
C02539=1029.217,296.685,373.679,170.938,46.211,158.926
C02540=1029.224,296.932,373.647,170.942,46.210,158.926
C02541=1029.231,297.180,373.615,170.946,46.210,158.926
C02542=1029.237,297.428,373.583,170.951,46.210,158.927
C02543=1029.244,297.676,373.550,170.955,46.209,158.927
C02544=1029.251,297.924,373.517,170.959,46.209,158.928
C02545=1029.257,298.171,373.485,170.965,46.208,158.928
C02546=1029.264,298.419,373.452,170.969,46.208,158.929
C02547=1029.271,298.667,373.419,170.973,46.208,158.929
C02548=1029.277,298.915,373.387,170.978,46.207,158.929
C02549=1029.285,299.162,373.353,170.982,46.207,158.930
C02550=1029.291,299.409,373.321,170.986,46.206,158.930
C02551=1029.298,299.658,373.287,170.990,46.206,158.931
C02552=1029.304,299.905,373.255,170.996,46.206,158.931
C02553=1029.311,300.153,373.223,171.000,46.206,158.932
C02554=1029.318,300.401,373.189,171.005,46.205,158.932
C02555=1029.325,300.649,373.157,171.009,46.205,158.932
C02556=1029.332,300.897,373.124,171.013,46.204,158.933
C02557=1029.339,301.144,373.091,171.018,46.204,158.933
C02558=1029.346,301.392,373.058,171.023,46.203,158.934
C02559=1029.353,301.639,373.025,171.028,46.204,158.934
C02560=1029.359,301.887,372.993,171.032,46.203,158.935
C02561=1029.366,302.135,372.960,171.036,46.203,158.935
C02562=1029.373,302.382,372.927,171.041,46.202,158.936
C02563=1029.380,302.630,372.894,171.046,46.202,158.936
C02564=1029.387,302.878,372.861,171.051,46.202,158.937
C02565=1029.393,303.126,372.828,171.055,46.202,158.937
C02566=1029.401,303.372,372.795,171.059,46.201,158.937
C02567=1029.408,303.621,372.762,171.065,46.201,158.938
C02568=1029.415,303.869,372.729,171.069,46.201,158.938
C02569=1029.422,304.116,372.696,171.073,46.200,158.939
C02570=1029.429,304.364,372.663,171.078,46.200,158.939
C02571=1029.435,304.612,372.630,171.083,46.200,158.940
C02572=1029.442,304.859,372.596,171.088,46.200,158.940
C02573=1029.449,305.107,372.564,171.092,46.199,158.941
C02574=1029.457,305.354,372.530,171.097,46.199,158.941
C02575=1029.463,305.603,372.497,171.102,46.199,158.942
C02576=1029.471,305.849,372.464,171.106,46.198,158.942
C02577=1029.482,306.263,372.409,171.114,46.198,158.943
C02578=1029.494,306.679,372.353,171.122,46.198,158.944
C02579=1029.506,307.092,372.297,171.129,46.197,158.945
C02580=1029.517,307.507,372.242,171.137,46.197,158.945
C02581=1029.524,307.754,372.208,171.143,46.197,158.946
C02582=1029.532,308.002,372.176,171.147,46.197,158.946
C02583=1029.539,308.249,372.143,171.152,46.197,158.947
C02584=1029.546,308.497,372.109,171.157,46.196,158.948
C02585=1029.554,308.745,372.076,171.162,46.196,158.948
C02586=1029.560,308.992,372.043,171.166,46.196,158.949
C02587=1029.567,309.240,372.009,171.172,46.196,158.949
C02588=1029.574,309.488,371.976,171.176,46.196,158.950
C02589=1029.582,309.735,371.943,171.180,46.196,158.950
C02590=1029.589,309.983,371.909,171.186,46.195,158.951
C02591=1029.596,310.230,371.875,171.190,46.195,158.951
C02592=1029.603,310.478,371.842,171.195,46.195,158.952
C02593=1029.611,310.726,371.809,171.200,46.195,158.952
C02594=1029.618,310.973,371.775,171.205,46.195,158.953
C02595=1029.625,311.220,371.742,171.209,46.195,158.953
C02596=1029.632,311.468,371.708,171.215,46.195,158.954
C02597=1029.638,311.716,371.673,171.219,46.195,158.954
C02598=1029.645,311.964,371.640,171.224,46.195,158.955
C02599=1029.651,312.211,371.606,171.229,46.195,158.956
C02600=1029.659,312.459,371.572,171.234,46.195,158.956
C02601=1029.666,312.706,371.538,171.239,46.195,158.957
C02602=1029.672,312.954,371.503,171.243,46.195,158.957
C02603=1029.679,313.201,371.469,171.249,46.195,158.958
C02604=1029.686,313.448,371.435,171.253,46.195,158.959
C02605=1029.693,313.696,371.401,171.258,46.196,158.959
C02606=1029.700,313.944,371.367,171.263,46.195,158.960
C02607=1029.707,314.192,371.333,171.268,46.195,158.960
C02608=1029.714,314.440,371.299,171.273,46.195,158.961
C02609=1029.721,314.686,371.265,171.278,46.195,158.961
C02610=1029.728,314.934,371.231,171.283,46.196,158.962
C02611=1029.734,315.182,371.197,171.287,46.196,158.963
C02612=1029.741,315.429,371.163,171.293,46.196,158.963
C02613=1029.749,315.676,371.128,171.298,46.196,158.964
C02614=1029.755,315.924,371.094,171.303,46.196,158.964
C02615=1029.763,316.172,371.060,171.308,46.196,158.965
C02616=1029.769,316.419,371.025,171.312,46.197,158.966
C02617=1029.777,316.667,370.991,171.318,46.196,158.966
C02618=1029.783,316.913,370.957,171.323,46.197,158.967
C02619=1029.790,317.161,370.922,171.327,46.197,158.967
C02620=1029.797,317.409,370.889,171.333,46.197,158.968
C02621=1029.805,317.656,370.854,171.338,46.197,158.969
C02622=1029.811,317.904,370.820,171.343,46.197,158.969
C02623=1029.819,318.151,370.785,171.348,46.197,158.970
C02624=1029.825,318.399,370.751,171.353,46.198,158.971
C02625=1029.833,318.646,370.716,171.358,46.198,158.971
C02626=1029.840,318.894,370.682,171.363,46.198,158.972
C02627=1029.847,319.142,370.647,171.368,46.198,158.972
C02628=1029.854,319.390,370.613,171.373,46.199,158.973
C02629=1029.861,319.637,370.578,171.379,46.199,158.974
C02630=1029.868,319.885,370.544,171.383,46.199,158.974
C02631=1029.876,320.132,370.509,171.388,46.200,158.975
C02632=1029.883,320.379,370.474,171.394,46.200,158.976
C02633=1029.888,320.588,370.446,171.398,46.200,158.976
C02634=1029.895,320.798,370.416,171.402,46.200,158.977
C02635=1029.901,321.008,370.387,171.406,46.200,158.977
C02636=1029.907,321.217,370.358,171.411,46.200,158.978
C02637=1029.913,321.427,370.328,171.416,46.200,158.978
C02638=1029.919,321.637,370.300,171.420,46.200,158.979
C02639=1029.926,321.846,370.270,171.424,46.201,158.979
C02640=1029.931,322.056,370.240,171.428,46.201,158.980
C02641=1029.939,322.303,370.206,171.434,46.201,158.981
C02642=1029.946,322.551,370.171,171.439,46.202,158.981
C02643=1029.953,322.799,370.137,171.444,46.202,158.982
C02644=1029.960,323.046,370.102,171.449,46.202,158.983
C02645=1029.968,323.294,370.067,171.455,46.203,158.983
C02646=1029.975,323.541,370.032,171.460,46.203,158.984
C02647=1029.983,323.788,369.997,171.465,46.203,158.985
C02648=1029.989,324.036,369.963,171.470,46.204,158.985
C02649=1029.997,324.283,369.928,171.476,46.204,158.986
C02650=1030.004,324.531,369.893,171.481,46.205,158.987
C02651=1030.011,324.778,369.858,171.486,46.204,158.988
C02652=1030.019,325.026,369.823,171.491,46.205,158.988
C02653=1030.026,325.273,369.788,171.497,46.205,158.989
C02654=1030.034,325.520,369.754,171.502,46.205,158.990
C02655=1030.041,325.768,369.718,171.507,46.206,158.990
C02656=1030.049,326.015,369.684,171.513,46.206,158.991
C02657=1030.055,326.263,369.649,171.518,46.207,158.992
C02658=1030.064,326.510,369.614,171.523,46.207,158.992
C02659=1030.070,326.758,369.579,171.528,46.208,158.993
C02660=1030.078,327.005,369.544,171.534,46.208,158.994
C02661=1030.086,327.252,369.509,171.540,46.208,158.995
C02662=1030.093,327.500,369.474,171.544,46.208,158.995
C02663=1030.101,327.748,369.439,171.550,46.209,158.996
C02664=1030.108,327.994,369.403,171.555,46.210,158.997
C02665=1030.115,328.242,369.368,171.561,46.210,158.997
C02666=1030.122,328.490,369.333,171.567,46.210,158.998
C02667=1030.129,328.737,369.297,171.572,46.211,158.999
C02668=1030.136,328.985,369.261,171.577,46.212,159.000
C02669=1030.144,329.232,369.227,171.582,46.212,159.000
C02670=1030.152,329.479,369.191,171.588,46.213,159.001
C02671=1030.158,329.726,369.155,171.593,46.213,159.002
C02672=1030.166,329.973,369.120,171.599,46.214,159.003
C02673=1030.173,330.221,369.084,171.605,46.214,159.004
C02674=1030.180,330.468,369.048,171.610,46.215,159.004
C02675=1030.187,330.716,369.013,171.615,46.215,159.005
C02676=1030.195,330.963,368.977,171.620,46.216,159.006
C02677=1030.203,331.211,368.942,171.626,46.217,159.007
C02678=1030.210,331.457,368.906,171.632,46.217,159.007
C02679=1030.217,331.705,368.871,171.637,46.218,159.008
C02680=1030.224,331.952,368.835,171.643,46.219,159.009
C02681=1030.231,332.200,368.799,171.649,46.219,159.010
C02682=1030.239,332.448,368.763,171.653,46.220,159.011
C02683=1030.246,332.694,368.727,171.659,46.221,159.011
C02684=1030.254,332.942,368.692,171.665,46.221,159.012
C02685=1030.261,333.189,368.656,171.670,46.222,159.013
C02686=1030.269,333.436,368.620,171.676,46.222,159.014
C02687=1030.276,333.684,368.585,171.682,46.223,159.015
C02688=1030.283,333.931,368.549,171.687,46.224,159.015
C02689=1030.291,334.179,368.513,171.693,46.224,159.016
C02690=1030.298,334.425,368.477,171.699,46.225,159.017
C02691=1030.306,334.673,368.441,171.704,46.226,159.018
C02692=1030.314,334.920,368.404,171.710,46.227,159.019
C02693=1030.325,335.335,368.345,171.719,46.228,159.020
C02694=1030.337,335.750,368.284,171.729,46.229,159.021
C02695=1030.350,336.165,368.223,171.739,46.231,159.023
C02696=1030.362,336.580,368.162,171.748,46.232,159.024
C02697=1030.369,336.826,368.126,171.753,46.233,159.025
C02698=1030.377,337.073,368.089,171.759,46.234,159.026
C02699=1030.385,337.321,368.053,171.765,46.234,159.027
C02700=1030.393,337.568,368.017,171.770,46.236,159.028
C02701=1030.400,337.815,367.981,171.776,46.236,159.029
C02702=1030.407,338.063,367.944,171.782,46.237,159.029
C02703=1030.414,338.310,367.908,171.788,46.238,159.030
C02704=1030.422,338.557,367.872,171.793,46.239,159.031
C02705=1030.430,338.805,367.836,171.799,46.240,159.032
C02706=1030.438,339.052,367.799,171.805,46.240,159.033
C02707=1030.445,339.298,367.763,171.811,46.241,159.034
C02708=1030.452,339.546,367.726,171.817,46.242,159.035
C02709=1030.459,339.794,367.690,171.822,46.243,159.036
C02710=1030.467,340.040,367.653,171.828,46.244,159.037
C02711=1030.475,340.288,367.617,171.834,46.245,159.037
C02712=1030.483,340.535,367.580,171.841,46.246,159.038
C02713=1030.490,340.782,367.543,171.846,46.246,159.039
C02714=1030.498,341.030,367.507,171.852,46.248,159.040
C02715=1030.505,341.276,367.470,171.858,46.249,159.041
C02716=1030.512,341.524,367.433,171.864,46.250,159.042
C02717=1030.520,341.771,367.396,171.870,46.251,159.043
C02718=1030.528,342.018,367.360,171.876,46.252,159.044
C02719=1030.535,342.265,367.323,171.881,46.253,159.045
C02720=1030.542,342.513,367.286,171.887,46.254,159.046
C02721=1030.550,342.760,367.249,171.893,46.255,159.047
C02722=1030.558,343.007,367.212,171.900,46.256,159.048
C02723=1030.565,343.254,367.176,171.905,46.257,159.048
C02724=1030.573,343.501,367.138,171.912,46.258,159.049
C02725=1030.581,343.748,367.101,171.918,46.259,159.050
C02726=1030.588,343.996,367.065,171.923,46.260,159.051
C02727=1030.596,344.243,367.028,171.929,46.262,159.052
C02728=1030.603,344.490,366.990,171.935,46.263,159.053
C02729=1030.611,344.737,366.953,171.941,46.263,159.054
C02730=1030.618,344.984,366.916,171.948,46.264,159.055
C02731=1030.626,345.231,366.879,171.954,46.265,159.056
C02732=1030.633,345.478,366.842,171.960,46.267,159.057
C02733=1030.641,345.725,366.805,171.966,46.268,159.058
C02734=1030.649,345.973,366.767,171.972,46.269,159.059
C02735=1030.657,346.220,366.730,171.977,46.270,159.060
C02736=1030.664,346.467,366.693,171.984,46.271,159.061
C02737=1030.672,346.714,366.656,171.990,46.273,159.062
C02738=1030.679,346.961,366.618,171.996,46.274,159.063
C02739=1030.687,347.208,366.581,172.002,46.275,159.064
C02740=1030.694,347.455,366.544,172.008,46.276,159.065
C02741=1030.703,347.702,366.506,172.015,46.277,159.066
C02742=1030.710,347.949,366.469,172.021,46.278,159.067
C02743=1030.718,348.196,366.432,172.027,46.280,159.068
C02744=1030.725,348.443,366.394,172.034,46.281,159.069
C02745=1030.734,348.691,366.357,172.040,46.282,159.070
C02746=1030.741,348.938,366.320,172.046,46.284,159.071
C02747=1030.749,349.185,366.281,172.052,46.285,159.072
C02748=1030.757,349.431,366.244,172.059,46.286,159.074
C02749=1030.770,349.843,366.181,172.069,46.289,159.075
C02750=1030.782,350.255,366.119,172.080,46.291,159.077
C02751=1030.795,350.666,366.056,172.090,46.293,159.079
C02752=1030.808,351.078,365.992,172.100,46.296,159.081
C02753=1030.816,351.325,365.955,172.106,46.297,159.082
C02754=1030.824,351.571,365.917,172.113,46.298,159.083
C02755=1030.831,351.819,365.879,172.119,46.300,159.084
C02756=1030.839,352.066,365.841,172.125,46.301,159.085
C02757=1030.847,352.312,365.804,172.133,46.302,159.086
C02758=1030.855,352.560,365.765,172.139,46.303,159.087
C02759=1030.862,352.807,365.728,172.146,46.305,159.088
C02760=1030.870,353.054,365.689,172.152,46.306,159.089
C02761=1030.878,353.300,365.651,172.158,46.308,159.090
C02762=1030.886,353.547,365.614,172.164,46.309,159.091
C02763=1030.894,353.795,365.575,172.171,46.311,159.093
C02764=1030.902,354.041,365.537,172.177,46.312,159.094
C02765=1030.910,354.289,365.499,172.184,46.314,159.095
C02766=1030.917,354.535,365.461,172.190,46.315,159.096
C02767=1030.926,354.782,365.423,172.198,46.317,159.097
C02768=1030.934,355.029,365.385,172.204,46.318,159.098
C02769=1030.942,355.276,365.346,172.210,46.320,159.099
C02770=1030.949,355.523,365.309,172.217,46.321,159.101
C02771=1030.957,355.770,365.270,172.223,46.323,159.102
C02772=1030.965,356.018,365.231,172.229,46.324,159.103
C02773=1030.973,356.264,365.193,172.236,46.326,159.104
C02774=1030.981,356.511,365.155,172.243,46.327,159.105
C02775=1030.989,356.758,365.116,172.250,46.329,159.106
C02776=1030.997,357.005,365.078,172.256,46.331,159.107
C02777=1031.004,357.252,365.040,172.263,46.333,159.109
C02778=1031.012,357.499,365.001,172.269,46.334,159.110
C02779=1031.021,357.746,364.962,172.277,46.336,159.111
C02780=1031.028,357.992,364.923,172.283,46.337,159.112
C02781=1031.037,358.239,364.885,172.290,46.339,159.113
C02782=1031.045,358.486,364.846,172.296,46.340,159.114
C02783=1031.052,358.733,364.808,172.303,46.343,159.116
C02784=1031.060,358.980,364.769,172.310,46.344,159.117
C02785=1031.069,359.227,364.730,172.317,46.346,159.118
C02786=1031.076,359.473,364.692,172.323,46.347,159.119
C02787=1031.085,359.720,364.653,172.330,46.349,159.121
C02788=1031.093,359.967,364.614,172.337,46.351,159.122
C02789=1031.101,360.214,364.575,172.344,46.352,159.123
C02790=1031.109,360.461,364.537,172.350,46.354,159.124
C02791=1031.117,360.707,364.498,172.358,46.356,159.126
C02792=1031.125,360.955,364.459,172.365,46.358,159.127
C02793=1031.134,361.201,364.420,172.371,46.360,159.128
C02794=1031.141,361.449,364.380,172.378,46.361,159.129
C02795=1031.149,361.695,364.342,172.385,46.363,159.131
C02796=1031.157,361.942,364.303,172.392,46.365,159.132
C02797=1031.166,362.188,364.264,172.398,46.367,159.133
C02798=1031.173,362.435,364.224,172.406,46.369,159.134
C02799=1031.182,362.682,364.185,172.413,46.370,159.136
C02800=1031.190,362.929,364.146,172.420,46.373,159.137
C02801=1031.197,363.175,364.106,172.427,46.374,159.138
C02802=1031.206,363.422,364.067,172.434,46.376,159.140
C02803=1031.214,363.669,364.028,172.440,46.378,159.141
C02804=1031.221,363.916,363.988,172.448,46.380,159.142
C02805=1031.236,364.333,363.922,172.460,46.383,159.144
C02806=1031.250,364.751,363.855,172.472,46.387,159.147
C02807=1031.263,365.169,363.788,172.483,46.390,159.149
C02808=1031.278,365.587,363.721,172.495,46.394,159.151
C02809=1031.285,365.834,363.681,172.503,46.396,159.153
C02810=1031.294,366.080,363.642,172.510,46.397,159.154
C02811=1031.302,366.327,363.602,172.517,46.400,159.155
C02812=1031.310,366.574,363.563,172.524,46.402,159.157
C02813=1031.318,366.821,363.523,172.531,46.404,159.158
C02814=1031.327,367.067,363.484,172.539,46.405,159.159
C02815=1031.335,367.314,363.444,172.545,46.408,159.161
C02816=1031.343,367.560,363.404,172.553,46.410,159.162
C02817=1031.352,367.807,363.365,172.560,46.412,159.163
C02818=1031.360,368.053,363.325,172.568,46.414,159.165
C02819=1031.369,368.301,363.285,172.575,46.416,159.166
C02820=1031.377,368.547,363.245,172.582,46.418,159.168
C02821=1031.385,368.794,363.205,172.589,46.420,159.169
C02822=1031.394,369.040,363.166,172.597,46.422,159.170
C02823=1031.403,369.287,363.125,172.605,46.425,159.172
C02824=1031.411,369.534,363.085,172.612,46.427,159.173
C02825=1031.419,369.780,363.045,172.620,46.429,159.175
C02826=1031.427,370.027,363.005,172.626,46.431,159.176
C02827=1031.435,370.273,362.965,172.634,46.433,159.177
C02828=1031.443,370.521,362.925,172.641,46.435,159.179
C02829=1031.452,370.767,362.884,172.649,46.438,159.180
C02830=1031.460,371.013,362.844,172.656,46.440,159.182
C02831=1031.468,371.260,362.804,172.664,46.442,159.183
C02832=1031.477,371.506,362.764,172.672,46.445,159.185
C02833=1031.485,371.753,362.723,172.679,46.447,159.186
C02834=1031.493,372.000,362.683,172.686,46.449,159.188
C02835=1031.502,372.246,362.643,172.693,46.452,159.189
C02836=1031.511,372.493,362.602,172.701,46.454,159.191
C02837=1031.519,372.739,362.561,172.709,46.456,159.192
C02838=1031.528,372.986,362.521,172.716,46.459,159.194
C02839=1031.536,373.232,362.480,172.724,46.461,159.195
C02840=1031.545,373.479,362.439,172.732,46.463,159.197
C02841=1031.553,373.725,362.399,172.739,46.466,159.198
C02842=1031.561,373.971,362.359,172.747,46.468,159.200
C02843=1031.570,374.218,362.318,172.755,46.470,159.201
C02844=1031.579,374.464,362.278,172.763,46.473,159.203
C02845=1031.587,374.711,362.237,172.770,46.476,159.204
C02846=1031.595,374.957,362.196,172.778,46.478,159.206
C02847=1031.604,375.204,362.155,172.786,46.480,159.207
C02848=1031.613,375.451,362.115,172.793,46.483,159.209
C02849=1031.621,375.697,362.074,172.801,46.485,159.210
C02850=1031.630,375.944,362.033,172.809,46.488,159.212
C02851=1031.639,376.190,361.992,172.817,46.490,159.214
C02852=1031.648,376.437,361.951,172.825,46.493,159.215
C02853=1031.656,376.683,361.910,172.832,46.495,159.217
C02854=1031.665,376.930,361.870,172.840,46.498,159.218
C02855=1031.674,377.176,361.828,172.848,46.500,159.220
C02856=1031.682,377.422,361.788,172.856,46.503,159.221
C02857=1031.691,377.669,361.747,172.864,46.505,159.223
C02858=1031.700,377.916,361.705,172.873,46.508,159.225
C02859=1031.708,378.161,361.664,172.880,46.511,159.226
C02860=1031.717,378.408,361.623,172.888,46.513,159.228
C02861=1031.724,378.627,361.586,172.895,46.515,159.229
C02862=1031.732,378.847,361.549,172.903,46.518,159.231
C02863=1031.740,379.066,361.512,172.910,46.520,159.232
C02864=1031.748,379.285,361.475,172.917,46.523,159.234
C02865=1031.755,379.504,361.438,172.923,46.525,159.235
C02866=1031.763,379.724,361.401,172.931,46.527,159.237
C02867=1031.771,379.943,361.365,172.938,46.530,159.238
C02868=1031.778,380.163,361.328,172.945,46.532,159.240
C02869=1031.787,380.409,361.286,172.954,46.535,159.241
C02870=1031.796,380.656,361.244,172.962,46.538,159.243
C02871=1031.805,380.902,361.202,172.970,46.540,159.245
C02872=1031.813,381.148,361.161,172.978,46.544,159.246
C02873=1031.822,381.394,361.119,172.986,46.546,159.248
C02874=1031.831,381.640,361.078,172.995,46.549,159.250
C02875=1031.840,381.887,361.036,173.003,46.552,159.251
C02876=1031.849,382.133,360.994,173.011,46.554,159.253
C02877=1031.858,382.379,360.953,173.020,46.557,159.255
C02878=1031.867,382.626,360.911,173.028,46.560,159.257
C02879=1031.876,382.872,360.869,173.036,46.563,159.258
C02880=1031.885,383.119,360.827,173.045,46.566,159.260
C02881=1031.894,383.365,360.786,173.053,46.569,159.262
C02882=1031.903,383.611,360.744,173.061,46.572,159.264
C02883=1031.912,383.857,360.701,173.069,46.574,159.265
C02884=1031.921,384.103,360.660,173.078,46.577,159.267
C02885=1031.930,384.350,360.618,173.086,46.581,159.269
C02886=1031.939,384.595,360.576,173.094,46.584,159.271
C02887=1031.947,384.842,360.533,173.103,46.586,159.272
C02888=1031.956,385.089,360.492,173.112,46.589,159.274
C02889=1031.965,385.334,360.449,173.120,46.592,159.276
C02890=1031.974,385.581,360.407,173.129,46.595,159.278
C02891=1031.984,385.827,360.365,173.137,46.598,159.280
C02892=1031.993,386.073,360.323,173.146,46.601,159.281
C02893=1032.002,386.319,360.281,173.154,46.605,159.283
C02894=1032.011,386.566,360.239,173.164,46.607,159.285
C02895=1032.021,386.811,360.196,173.172,46.611,159.287
C02896=1032.030,387.058,360.154,173.181,46.614,159.289
C02897=1032.039,387.304,360.111,173.189,46.617,159.291
C02898=1032.048,387.550,360.069,173.197,46.620,159.292
C02899=1032.057,387.796,360.026,173.207,46.623,159.294
C02900=1032.066,388.043,359.983,173.215,46.626,159.296
C02901=1032.075,388.289,359.941,173.224,46.629,159.298
C02902=1032.084,388.535,359.899,173.232,46.632,159.300
C02903=1032.093,388.782,359.855,173.242,46.635,159.302
C02904=1032.103,389.027,359.813,173.251,46.639,159.304
C02905=1032.112,389.273,359.771,173.259,46.642,159.306
C02906=1032.122,389.519,359.728,173.269,46.645,159.308
C02907=1032.130,389.766,359.685,173.277,46.648,159.310
C02908=1032.139,390.011,359.642,173.286,46.652,159.311
C02909=1032.149,390.257,359.598,173.295,46.655,159.313
C02910=1032.158,390.503,359.556,173.304,46.658,159.315
C02911=1032.167,390.750,359.512,173.313,46.662,159.317
C02912=1032.176,390.996,359.470,173.322,46.665,159.319
C02913=1032.186,391.242,359.426,173.331,46.668,159.321
C02914=1032.195,391.488,359.383,173.340,46.672,159.323
C02915=1032.205,391.734,359.341,173.349,46.675,159.325
C02916=1032.214,391.979,359.297,173.358,46.678,159.327
C02917=1032.224,392.226,359.254,173.368,46.682,159.329
C02918=1032.232,392.471,359.210,173.376,46.685,159.331
C02919=1032.242,392.718,359.168,173.386,46.689,159.333
C02920=1032.251,392.963,359.124,173.395,46.692,159.335
C02921=1032.260,393.201,359.082,173.403,46.695,159.337
C02922=1032.269,393.437,359.040,173.413,46.699,159.339
C02923=1032.279,393.675,358.998,173.421,46.702,159.341
C02924=1032.287,393.911,358.956,173.430,46.705,159.343
C02925=1032.297,394.149,358.914,173.439,46.709,159.345
C02926=1032.306,394.385,358.873,173.449,46.712,159.347
C02927=1032.315,394.623,358.831,173.457,46.715,159.349
C02928=1032.324,394.859,358.789,173.466,46.719,159.351
C02929=1032.333,395.105,358.745,173.476,46.722,159.353
C02930=1032.343,395.352,358.701,173.486,46.726,159.355
C02931=1032.352,395.597,358.658,173.495,46.730,159.357
C02932=1032.362,395.843,358.614,173.504,46.733,159.359
C02933=1032.371,396.089,358.570,173.513,46.737,159.362
C02934=1032.381,396.335,358.526,173.523,46.741,159.364
C02935=1032.391,396.581,358.482,173.533,46.744,159.366
C02936=1032.400,396.826,358.437,173.542,46.748,159.368
C02937=1032.410,397.072,358.394,173.552,46.751,159.370
C02938=1032.419,397.318,358.350,173.562,46.755,159.372
C02939=1032.429,397.564,358.306,173.571,46.759,159.374
C02940=1032.439,397.810,358.262,173.581,46.763,159.377
C02941=1032.449,398.055,358.217,173.591,46.766,159.379
C02942=1032.458,398.301,358.173,173.601,46.770,159.381
C02943=1032.468,398.547,358.130,173.610,46.774,159.383
C02944=1032.478,398.793,358.085,173.619,46.778,159.385
C02945=1032.487,399.039,358.041,173.630,46.781,159.388
C02946=1032.497,399.284,357.996,173.640,46.785,159.390
C02947=1032.506,399.530,357.952,173.650,46.789,159.392
C02948=1032.517,399.776,357.908,173.659,46.793,159.394
C02949=1032.526,400.022,357.864,173.669,46.797,159.397
C02950=1032.536,400.267,357.819,173.679,46.801,159.399
C02951=1032.546,400.513,357.774,173.689,46.805,159.401
C02952=1032.556,400.760,357.729,173.699,46.809,159.403
C02953=1032.565,401.005,357.685,173.709,46.813,159.406
C02954=1032.575,401.251,357.640,173.719,46.817,159.408
C02955=1032.585,401.496,357.595,173.728,46.821,159.410
C02956=1032.595,401.742,357.550,173.739,46.825,159.412
C02957=1032.605,401.988,357.505,173.749,46.828,159.415
C02958=1032.615,402.233,357.460,173.759,46.833,159.417
C02959=1032.624,402.479,357.415,173.769,46.837,159.420
C02960=1032.634,402.724,357.370,173.779,46.841,159.422
C02961=1032.644,402.971,357.325,173.790,46.845,159.424
C02962=1032.654,403.216,357.280,173.800,46.849,159.427
C02963=1032.664,403.462,357.236,173.810,46.853,159.429
C02964=1032.674,403.708,357.190,173.820,46.857,159.431
C02965=1032.684,403.953,357.145,173.831,46.862,159.434
C02966=1032.694,404.198,357.100,173.841,46.866,159.436
C02967=1032.704,404.445,357.055,173.851,46.870,159.439
C02968=1032.713,404.690,357.009,173.862,46.874,159.441
C02969=1032.724,404.936,356.964,173.873,46.878,159.444
C02970=1032.734,405.181,356.918,173.883,46.882,159.446
C02971=1032.744,405.427,356.873,173.894,46.887,159.448
C02972=1032.754,405.672,356.827,173.904,46.891,159.451
C02973=1032.764,405.918,356.782,173.914,46.895,159.453
C02974=1032.774,406.163,356.737,173.925,46.900,159.456
C02975=1032.784,406.410,356.691,173.936,46.904,159.458
C02976=1032.795,406.655,356.645,173.947,46.908,159.461
C02977=1032.805,406.900,356.599,173.957,46.913,159.463
C02978=1032.815,407.146,356.553,173.968,46.917,159.466
C02979=1032.826,407.392,356.508,173.979,46.921,159.468
C02980=1032.836,407.637,356.463,173.989,46.925,159.471
C02981=1032.846,407.886,356.416,174.000,46.930,159.473
C02982=1032.857,408.136,356.370,174.012,46.934,159.476
C02983=1032.867,408.384,356.323,174.022,46.939,159.479
C02984=1032.877,408.634,356.276,174.034,46.943,159.481
C02985=1032.888,408.879,356.230,174.044,46.948,159.484
C02986=1032.899,409.125,356.184,174.055,46.952,159.486
C02987=1032.909,409.370,356.138,174.066,46.957,159.489
C02988=1032.919,409.615,356.093,174.077,46.961,159.491
C02989=1032.930,409.861,356.047,174.089,46.966,159.494
C02990=1032.940,410.106,355.999,174.099,46.970,159.497
C02991=1032.951,410.352,355.954,174.111,46.975,159.499
C02992=1032.961,410.597,355.908,174.122,46.980,159.502
C02993=1032.972,410.843,355.862,174.133,46.984,159.505
C02994=1032.982,411.088,355.815,174.144,46.989,159.507
C02995=1032.993,411.334,355.769,174.156,46.993,159.510
C02996=1033.003,411.579,355.721,174.166,46.998,159.513
C02997=1033.014,411.825,355.676,174.178,47.003,159.516
C02998=1033.024,412.071,355.628,174.189,47.008,159.518
C02999=1033.035,412.316,355.581,174.201,47.012,159.521
C03000=1033.045,412.562,355.535,174.211,47.017,159.524
C03001=1033.056,412.807,355.488,174.223,47.022,159.526
C03002=1033.066,413.052,355.441,174.235,47.026,159.529
C03003=1033.077,413.297,355.394,174.246,47.032,159.532
C03004=1033.087,413.542,355.347,174.258,47.036,159.535
C03005=1033.099,413.788,355.300,174.270,47.041,159.538
C03006=1033.109,414.034,355.254,174.281,47.045,159.540
C03007=1033.120,414.279,355.207,174.293,47.051,159.543
C03008=1033.132,414.524,355.159,174.304,47.055,159.546
C03009=1033.142,414.769,355.112,174.316,47.061,159.549
C03010=1033.153,415.014,355.065,174.328,47.065,159.552
C03011=1033.163,415.260,355.018,174.340,47.070,159.555
C03012=1033.174,415.505,354.971,174.351,47.075,159.557
C03013=1033.185,415.750,354.924,174.363,47.080,159.560
C03014=1033.196,415.995,354.876,174.375,47.085,159.563
C03015=1033.207,416.240,354.829,174.387,47.090,159.566
C03016=1033.218,416.486,354.782,174.399,47.095,159.569
C03017=1033.229,416.732,354.734,174.411,47.100,159.572
C03018=1033.239,416.977,354.687,174.423,47.105,159.575
C03019=1033.251,417.222,354.639,174.436,47.110,159.578
C03020=1033.261,417.467,354.592,174.448,47.115,159.581
C03021=1033.273,417.713,354.543,174.460,47.120,159.584
C03022=1033.283,417.957,354.496,174.472,47.126,159.587
C03023=1033.295,418.203,354.449,174.484,47.131,159.590
C03024=1033.306,418.448,354.400,174.496,47.136,159.593
C03025=1033.316,418.693,354.352,174.509,47.141,159.596
C03026=1033.327,418.938,354.304,174.521,47.146,159.599
C03027=1033.338,419.184,354.256,174.533,47.152,159.602
C03028=1033.350,419.428,354.208,174.545,47.157,159.605
C03029=1033.361,419.673,354.160,174.559,47.162,159.608
C03030=1033.372,419.919,354.112,174.571,47.167,159.611
C03031=1033.383,420.164,354.063,174.583,47.173,159.614
C03032=1033.395,420.409,354.016,174.595,47.178,159.617
C03033=1033.406,420.654,353.967,174.609,47.183,159.620
C03034=1033.416,420.899,353.920,174.621,47.189,159.624
C03035=1033.428,421.144,353.871,174.634,47.195,159.627
C03036=1033.439,421.389,353.822,174.647,47.200,159.630
C03037=1033.451,421.634,353.775,174.659,47.205,159.633
C03038=1033.462,421.879,353.725,174.672,47.211,159.636
C03039=1033.473,422.124,353.677,174.685,47.216,159.639
C03040=1033.485,422.369,353.628,174.698,47.221,159.643
C03041=1033.504,422.764,353.550,174.719,47.230,159.648
C03042=1033.522,423.159,353.471,174.740,47.239,159.653
C03043=1033.540,423.554,353.393,174.761,47.248,159.658
C03044=1033.559,423.948,353.313,174.782,47.257,159.664
C03045=1033.570,424.193,353.264,174.795,47.263,159.667
C03046=1033.582,424.438,353.215,174.809,47.269,159.670
C03047=1033.593,424.683,353.166,174.822,47.274,159.674
C03048=1033.605,424.928,353.117,174.835,47.280,159.677
C03049=1033.617,425.173,353.068,174.849,47.286,159.680
C03050=1033.628,425.418,353.019,174.862,47.291,159.684
C03051=1033.640,425.663,352.970,174.875,47.298,159.687
C03052=1033.652,425.907,352.920,174.889,47.303,159.691
C03053=1033.663,426.152,352.871,174.903,47.309,159.694
C03054=1033.675,426.397,352.821,174.917,47.315,159.697
C03055=1033.687,426.641,352.772,174.931,47.321,159.701
C03056=1033.699,426.887,352.722,174.943,47.327,159.704
C03057=1033.710,427.131,352.673,174.957,47.332,159.708
C03058=1033.722,427.376,352.623,174.971,47.338,159.711
C03059=1033.735,427.621,352.573,174.985,47.344,159.715
C03060=1033.747,427.865,352.523,174.999,47.350,159.718
C03061=1033.758,428.111,352.473,175.013,47.356,159.722
C03062=1033.770,428.355,352.424,175.027,47.362,159.725
C03063=1033.782,428.600,352.374,175.041,47.368,159.729
C03064=1033.793,428.845,352.323,175.055,47.374,159.732
C03065=1033.805,429.089,352.273,175.069,47.380,159.736
C03066=1033.817,429.334,352.223,175.083,47.387,159.740
C03067=1033.830,429.579,352.173,175.097,47.392,159.743
C03068=1033.841,429.823,352.123,175.112,47.398,159.747
C03069=1033.853,430.068,352.072,175.127,47.405,159.751
C03070=1033.866,430.312,352.022,175.141,47.411,159.754
C03071=1033.878,430.557,351.972,175.155,47.417,159.758
C03072=1033.890,430.802,351.921,175.169,47.423,159.762
C03073=1033.902,431.047,351.870,175.185,47.430,159.766
C03074=1033.914,431.291,351.820,175.199,47.436,159.769
C03075=1033.926,431.535,351.770,175.213,47.442,159.773
C03076=1033.938,431.780,351.719,175.228,47.448,159.777
C03077=1033.956,432.134,351.645,175.249,47.457,159.782
C03078=1033.974,432.487,351.572,175.271,47.467,159.788
C03079=1033.992,432.840,351.498,175.293,47.476,159.793
C03080=1034.010,433.195,351.425,175.313,47.485,159.799
C03081=1034.023,433.439,351.374,175.329,47.492,159.803
C03082=1034.036,433.683,351.323,175.345,47.498,159.807
C03083=1034.048,433.928,351.272,175.359,47.505,159.810
C03084=1034.061,434.172,351.221,175.375,47.511,159.814
C03085=1034.073,434.417,351.170,175.390,47.517,159.818
C03086=1034.086,434.661,351.118,175.405,47.524,159.822
C03087=1034.098,434.905,351.067,175.420,47.530,159.826
C03088=1034.111,435.150,351.015,175.436,47.537,159.830
C03089=1034.124,435.394,350.964,175.452,47.544,159.834
C03090=1034.136,435.639,350.912,175.466,47.550,159.838
C03091=1034.149,435.882,350.860,175.482,47.557,159.842
C03092=1034.162,436.127,350.810,175.498,47.564,159.846
C03093=1034.174,436.371,350.757,175.514,47.571,159.850
C03094=1034.188,436.616,350.706,175.529,47.577,159.854
C03095=1034.200,436.860,350.654,175.545,47.584,159.858
C03096=1034.213,437.104,350.601,175.561,47.591,159.863
C03097=1034.226,437.357,350.548,175.577,47.598,159.867
C03098=1034.239,437.610,350.494,175.594,47.605,159.871
C03099=1034.253,437.863,350.440,175.610,47.612,159.876
C03100=1034.266,438.116,350.386,175.628,47.619,159.880
C03101=1034.280,438.360,350.334,175.644,47.626,159.884
C03102=1034.292,438.604,350.282,175.659,47.633,159.888
C03103=1034.305,438.848,350.229,175.676,47.640,159.893
C03104=1034.319,439.092,350.177,175.693,47.647,159.897
C03105=1034.331,439.337,350.124,175.709,47.653,159.901
C03106=1034.345,439.581,350.072,175.725,47.661,159.905
C03107=1034.358,439.825,350.019,175.742,47.668,159.910
C03108=1034.371,440.069,349.966,175.758,47.674,159.914
C03109=1034.385,440.313,349.914,175.774,47.682,159.918
C03110=1034.398,440.557,349.861,175.792,47.689,159.923
C03111=1034.411,440.801,349.808,175.808,47.696,159.927
C03112=1034.425,441.045,349.755,175.825,47.703,159.932
C03113=1034.438,441.289,349.702,175.841,47.710,159.936
C03114=1034.450,441.534,349.649,175.859,47.717,159.940
C03115=1034.464,441.778,349.596,175.876,47.725,159.945
C03116=1034.478,442.021,349.543,175.893,47.732,159.949
C03117=1034.491,442.265,349.490,175.910,47.739,159.954
C03118=1034.504,442.509,349.436,175.928,47.746,159.959
C03119=1034.518,442.753,349.383,175.944,47.754,159.963
C03120=1034.531,442.997,349.330,175.962,47.761,159.968
C03121=1034.546,443.240,349.277,175.979,47.769,159.972
C03122=1034.559,443.484,349.224,175.997,47.776,159.977
C03123=1034.573,443.727,349.170,176.014,47.783,159.981
C03124=1034.586,443.970,349.116,176.032,47.790,159.986
C03125=1034.601,444.214,349.064,176.049,47.798,159.991
C03126=1034.616,444.456,349.012,176.067,47.805,159.995
C03127=1034.632,444.700,348.960,176.084,47.812,160.000
C03128=1034.647,444.944,348.908,176.103,47.819,160.005
C03129=1034.664,445.187,348.857,176.120,47.826,160.009
C03130=1034.681,445.431,348.807,176.139,47.833,160.014
C03131=1034.699,445.675,348.757,176.157,47.839,160.018
C03132=1034.717,445.920,348.707,176.175,47.846,160.023
C03133=1034.735,446.163,348.658,176.193,47.853,160.027
C03134=1034.754,446.407,348.609,176.211,47.860,160.032
C03135=1034.774,446.651,348.559,176.231,47.866,160.036
C03136=1034.795,446.896,348.512,176.249,47.872,160.041
C03137=1034.815,447.140,348.465,176.267,47.879,160.045
C03138=1034.836,447.384,348.417,176.286,47.884,160.050
C03139=1034.858,447.628,348.370,176.305,47.891,160.054
C03140=1034.881,447.873,348.324,176.324,47.897,160.059
C03141=1034.903,448.118,348.279,176.343,47.903,160.063
C03142=1034.926,448.362,348.233,176.362,47.908,160.067
C03143=1034.950,448.607,348.189,176.381,47.914,160.072
C03144=1034.975,448.853,348.143,176.400,47.920,160.076
C03145=1035.000,449.097,348.099,176.419,47.926,160.081
C03146=1035.025,449.343,348.055,176.439,47.931,160.085
C03147=1035.051,449.588,348.012,176.458,47.936,160.090
C03148=1035.078,449.833,347.969,176.478,47.941,160.094
C03149=1035.105,450.078,347.927,176.497,47.947,160.098
C03150=1035.132,450.324,347.885,176.517,47.952,160.103
C03151=1035.160,450.568,347.844,176.537,47.957,160.107
C03152=1035.189,450.814,347.802,176.557,47.962,160.111
C03153=1035.218,451.059,347.762,176.577,47.967,160.116
C03154=1035.247,451.305,347.721,176.597,47.972,160.120
C03155=1035.278,451.551,347.681,176.618,47.977,160.125
C03156=1035.308,451.796,347.642,176.637,47.982,160.129
C03157=1035.337,452.019,347.607,176.656,47.986,160.133
C03158=1035.366,452.243,347.571,176.674,47.991,160.137
C03159=1035.395,452.467,347.537,176.693,47.995,160.141
C03160=1035.425,452.689,347.503,176.711,47.999,160.144
C03161=1035.137,452.748,347.177,176.715,48.067,160.166
C03162=1035.109,452.538,347.208,176.697,48.064,160.163
C03163=1035.082,452.328,347.241,176.679,48.060,160.159
C03164=1035.054,452.117,347.274,176.662,48.055,160.155
C03165=1035.026,451.906,347.308,176.644,48.052,160.151
C03166=1034.996,451.660,347.346,176.625,48.047,160.147
C03167=1034.965,451.415,347.386,176.604,48.043,160.143
C03168=1034.936,451.169,347.427,176.584,48.038,160.138
C03169=1034.906,450.924,347.466,176.564,48.033,160.134
C03170=1034.877,450.679,347.508,176.544,48.028,160.130
C03171=1034.849,450.434,347.548,176.524,48.023,160.125
C03172=1034.822,450.188,347.590,176.504,48.017,160.121
C03173=1034.794,449.942,347.633,176.484,48.012,160.117
C03174=1034.767,449.697,347.675,176.464,48.007,160.112
C03175=1034.740,449.452,347.718,176.445,48.002,160.108
C03176=1034.716,449.207,347.761,176.425,47.997,160.103
C03177=1034.690,448.962,347.806,176.406,47.991,160.099
C03178=1034.666,448.717,347.849,176.387,47.985,160.095
C03179=1034.641,448.472,347.894,176.367,47.980,160.090
C03180=1034.617,448.227,347.940,176.348,47.974,160.086
C03181=1034.594,447.983,347.985,176.329,47.969,160.081
C03182=1034.571,447.738,348.032,176.311,47.962,160.077
C03183=1034.550,447.494,348.078,176.291,47.956,160.072
C03184=1034.528,447.249,348.125,176.272,47.951,160.068
C03185=1034.507,447.005,348.172,176.254,47.944,160.063
C03186=1034.487,446.760,348.220,176.236,47.938,160.059
C03187=1034.467,446.517,348.268,176.217,47.932,160.054
C03188=1034.447,446.272,348.317,176.198,47.926,160.050
C03189=1034.428,446.028,348.366,176.180,47.919,160.045
C03190=1034.410,445.784,348.416,176.162,47.913,160.041
C03191=1034.392,445.540,348.465,176.143,47.906,160.036
C03192=1034.374,445.297,348.516,176.126,47.899,160.032
C03193=1034.358,445.053,348.566,176.107,47.892,160.027
C03194=1034.341,444.809,348.618,176.089,47.886,160.023
C03195=1034.325,444.565,348.669,176.072,47.879,160.018
C03196=1034.310,444.322,348.721,176.054,47.872,160.014
C03197=1034.295,444.079,348.774,176.035,47.865,160.009
C03198=1034.281,443.836,348.826,176.018,47.858,160.004
C03199=1034.268,443.593,348.880,176.000,47.850,160.000
C03200=1034.253,443.350,348.933,175.983,47.843,159.995
C03201=1034.240,443.106,348.987,175.966,47.836,159.991
C03202=1034.226,442.863,349.040,175.948,47.828,159.986
C03203=1034.212,442.618,349.093,175.931,47.821,159.981
C03204=1034.199,442.374,349.147,175.913,47.814,159.977
C03205=1034.186,442.130,349.199,175.896,47.807,159.972
C03206=1034.172,441.887,349.253,175.880,47.800,159.968
C03207=1034.158,441.642,349.307,175.862,47.792,159.963
C03208=1034.145,441.399,349.359,175.845,47.785,159.959
C03209=1034.131,441.155,349.413,175.828,47.778,159.954
C03210=1034.119,440.910,349.465,175.811,47.771,159.950
C03211=1034.105,440.666,349.518,175.794,47.764,159.945
C03212=1034.092,440.422,349.571,175.778,47.757,159.941
C03213=1034.079,440.178,349.624,175.761,47.750,159.937
C03214=1034.065,439.934,349.676,175.744,47.743,159.932
C03215=1034.052,439.690,349.729,175.727,47.737,159.928
C03216=1034.039,439.446,349.782,175.711,47.729,159.924
C03217=1034.025,439.202,349.834,175.695,47.723,159.920
C03218=1034.013,438.958,349.886,175.678,47.716,159.915
C03219=1034.000,438.714,349.938,175.662,47.709,159.911
C03220=1033.987,438.470,349.991,175.646,47.702,159.907
C03221=1033.973,438.226,350.043,175.630,47.695,159.903
C03222=1033.960,437.971,350.098,175.613,47.688,159.898
C03223=1033.946,437.718,350.152,175.595,47.681,159.894
C03224=1033.933,437.463,350.206,175.579,47.674,159.889
C03225=1033.920,437.209,350.261,175.562,47.667,159.885
C03226=1033.906,436.965,350.313,175.546,47.660,159.881
C03227=1033.895,436.720,350.364,175.530,47.653,159.877
C03228=1033.881,436.476,350.416,175.515,47.647,159.873
C03229=1033.869,436.232,350.468,175.499,47.640,159.869
C03230=1033.856,435.987,350.519,175.483,47.634,159.865
C03231=1033.843,435.743,350.571,175.467,47.627,159.861
C03232=1033.830,435.498,350.622,175.452,47.621,159.857
C03233=1033.817,435.255,350.674,175.437,47.614,159.853
C03234=1033.805,435.010,350.725,175.421,47.607,159.849
C03235=1033.792,434.766,350.777,175.406,47.601,159.845
C03236=1033.780,434.522,350.829,175.390,47.594,159.841
C03237=1033.767,434.277,350.880,175.375,47.588,159.837
C03238=1033.755,434.032,350.931,175.360,47.581,159.833
C03239=1033.742,433.788,350.982,175.344,47.575,159.829
C03240=1033.730,433.544,351.033,175.329,47.569,159.825
C03241=1033.716,433.299,351.084,175.315,47.562,159.821
C03242=1033.705,433.054,351.136,175.299,47.556,159.817
C03243=1033.692,432.810,351.186,175.285,47.550,159.814
C03244=1033.679,432.566,351.237,175.269,47.544,159.810
C03245=1033.667,432.321,351.287,175.255,47.537,159.806
C03246=1033.655,432.077,351.339,175.239,47.531,159.802
C03247=1033.643,431.832,351.389,175.225,47.525,159.798
C03248=1033.630,431.588,351.440,175.210,47.519,159.795
C03249=1033.618,431.343,351.490,175.196,47.513,159.791
C03250=1033.606,431.098,351.541,175.180,47.506,159.787
C03251=1033.593,430.854,351.592,175.166,47.500,159.783
C03252=1033.581,430.609,351.642,175.152,47.494,159.780
C03253=1033.569,430.364,351.692,175.137,47.488,159.776
C03254=1033.557,430.120,351.743,175.123,47.482,159.772
C03255=1033.545,429.875,351.794,175.108,47.476,159.769
C03256=1033.533,429.631,351.843,175.094,47.470,159.765
C03257=1033.521,429.386,351.893,175.080,47.464,159.761
C03258=1033.509,429.141,351.944,175.065,47.458,159.758
C03259=1033.497,428.896,351.994,175.051,47.452,159.754
C03260=1033.485,428.652,352.044,175.037,47.446,159.750
C03261=1033.473,428.407,352.094,175.023,47.440,159.747
C03262=1033.461,428.162,352.145,175.009,47.434,159.743
C03263=1033.449,427.918,352.194,174.995,47.428,159.740
C03264=1033.437,427.673,352.244,174.981,47.422,159.736
C03265=1033.426,427.428,352.293,174.967,47.417,159.733
C03266=1033.414,427.183,352.344,174.953,47.410,159.729
C03267=1033.403,426.938,352.393,174.939,47.405,159.726
C03268=1033.390,426.694,352.443,174.925,47.399,159.722
C03269=1033.378,426.448,352.493,174.912,47.393,159.719
C03270=1033.367,426.221,352.539,174.899,47.388,159.716
C03271=1033.357,425.994,352.584,174.887,47.383,159.713
C03272=1033.346,425.767,352.630,174.874,47.377,159.709
C03273=1033.334,425.540,352.675,174.862,47.372,159.706
C03274=1033.323,425.313,352.721,174.849,47.367,159.703
C03275=1033.313,425.085,352.767,174.837,47.361,159.700
C03276=1033.302,424.858,352.813,174.823,47.356,159.697
C03277=1033.291,424.631,352.858,174.811,47.351,159.694
C03278=1033.280,424.386,352.907,174.798,47.345,159.690
C03279=1033.268,424.141,352.956,174.785,47.340,159.687
C03280=1033.256,423.896,353.006,174.771,47.334,159.684
C03281=1033.245,423.651,353.055,174.759,47.328,159.680
C03282=1033.231,423.355,353.115,174.742,47.322,159.677
C03283=1033.218,423.059,353.173,174.727,47.315,159.673
C03284=1033.204,422.762,353.232,174.711,47.309,159.669
C03285=1033.190,422.466,353.291,174.695,47.302,159.665
C03286=1033.179,422.221,353.340,174.682,47.297,159.662
C03287=1033.167,421.976,353.388,174.670,47.291,159.658
C03288=1033.155,421.731,353.437,174.656,47.286,159.655
C03289=1033.144,421.486,353.485,174.644,47.280,159.652
C03290=1033.133,421.241,353.533,174.630,47.275,159.649
C03291=1033.122,420.996,353.582,174.618,47.270,159.646
C03292=1033.110,420.751,353.630,174.606,47.264,159.643
C03293=1033.099,420.505,353.678,174.592,47.259,159.639
C03294=1033.088,420.260,353.726,174.580,47.254,159.636
C03295=1033.077,420.015,353.775,174.567,47.249,159.633
C03296=1033.065,419.770,353.822,174.554,47.244,159.630
C03297=1033.054,419.525,353.870,174.542,47.238,159.627
C03298=1033.043,419.280,353.919,174.530,47.233,159.624
C03299=1033.032,419.034,353.967,174.517,47.228,159.621
C03300=1033.020,418.789,354.015,174.505,47.222,159.618
C03301=1033.010,418.544,354.063,174.492,47.218,159.615
C03302=1032.999,418.299,354.111,174.480,47.213,159.612
C03303=1032.988,418.054,354.159,174.468,47.208,159.609
C03304=1032.976,417.809,354.207,174.455,47.203,159.606
C03305=1032.966,417.563,354.254,174.443,47.197,159.603
C03306=1032.955,417.319,354.302,174.431,47.192,159.600
C03307=1032.944,417.073,354.350,174.419,47.187,159.597
C03308=1032.933,416.828,354.397,174.407,47.182,159.594
C03309=1032.922,416.582,354.445,174.395,47.177,159.591
C03310=1032.910,416.337,354.492,174.383,47.172,159.588
C03311=1032.900,416.092,354.540,174.371,47.167,159.585
C03312=1032.889,415.846,354.586,174.359,47.162,159.582
C03313=1032.878,415.602,354.634,174.347,47.157,159.579
C03314=1032.867,415.357,354.681,174.335,47.153,159.577
C03315=1032.856,415.111,354.729,174.323,47.148,159.574
C03316=1032.846,414.866,354.775,174.312,47.143,159.571
C03317=1032.835,414.620,354.823,174.300,47.138,159.568
C03318=1032.824,414.375,354.869,174.288,47.133,159.565
C03319=1032.814,414.130,354.917,174.276,47.129,159.562
C03320=1032.802,413.884,354.964,174.264,47.124,159.560
C03321=1032.792,413.639,355.011,174.253,47.119,159.557
C03322=1032.781,413.394,355.057,174.241,47.114,159.554
C03323=1032.771,413.148,355.105,174.230,47.109,159.551
C03324=1032.760,412.903,355.151,174.218,47.105,159.548
C03325=1032.749,412.657,355.199,174.207,47.100,159.546
C03326=1032.738,412.412,355.245,174.195,47.095,159.543
C03327=1032.728,412.167,355.292,174.183,47.091,159.540
C03328=1032.717,411.922,355.339,174.173,47.086,159.537
C03329=1032.707,411.676,355.385,174.161,47.081,159.535
C03330=1032.696,411.431,355.432,174.150,47.076,159.532
C03331=1032.687,411.185,355.478,174.138,47.072,159.529
C03332=1032.676,410.940,355.525,174.127,47.068,159.527
C03333=1032.666,410.694,355.571,174.116,47.063,159.524
C03334=1032.655,410.449,355.618,174.104,47.059,159.521
C03335=1032.644,410.203,355.664,174.094,47.054,159.519
C03336=1032.634,409.958,355.710,174.082,47.050,159.516
C03337=1032.623,409.712,355.756,174.071,47.045,159.513
C03338=1032.612,409.467,355.802,174.060,47.041,159.511
C03339=1032.601,409.222,355.848,174.049,47.036,159.508
C03340=1032.592,408.976,355.895,174.038,47.032,159.506
C03341=1032.581,408.730,355.941,174.027,47.028,159.503
C03342=1032.570,408.479,355.987,174.015,47.023,159.500
C03343=1032.560,408.227,356.034,174.005,47.019,159.498
C03344=1032.549,407.976,356.081,173.993,47.014,159.495
C03345=1032.539,407.725,356.128,173.983,47.010,159.493
C03346=1032.529,407.479,356.174,173.971,47.006,159.490
C03347=1032.518,407.234,356.220,173.961,47.001,159.488
C03348=1032.507,406.988,356.266,173.950,46.997,159.485
C03349=1032.498,406.743,356.310,173.939,46.993,159.483
C03350=1032.487,406.497,356.356,173.929,46.988,159.480
C03351=1032.476,406.251,356.402,173.918,46.984,159.478
C03352=1032.468,406.006,356.448,173.908,46.980,159.475
C03353=1032.457,405.760,356.494,173.896,46.976,159.473
C03354=1032.447,405.515,356.538,173.886,46.972,159.470
C03355=1032.437,405.269,356.584,173.876,46.967,159.468
C03356=1032.427,405.023,356.629,173.865,46.963,159.465
C03357=1032.416,404.778,356.675,173.855,46.959,159.463
C03358=1032.406,404.532,356.720,173.845,46.955,159.460
C03359=1032.396,404.287,356.766,173.833,46.951,159.458
C03360=1032.387,404.041,356.811,173.823,46.947,159.456
C03361=1032.377,403.795,356.856,173.813,46.942,159.453
C03362=1032.367,403.549,356.901,173.802,46.939,159.451
C03363=1032.357,403.304,356.947,173.792,46.934,159.448
C03364=1032.347,403.058,356.992,173.782,46.930,159.446
C03365=1032.337,402.813,357.037,173.772,46.927,159.444
C03366=1032.327,402.567,357.082,173.761,46.922,159.441
C03367=1032.317,402.322,357.126,173.751,46.918,159.439
C03368=1032.307,402.075,357.172,173.741,46.914,159.437
C03369=1032.297,401.830,357.216,173.731,46.911,159.434
C03370=1032.288,401.584,357.261,173.721,46.907,159.432
C03371=1032.278,401.339,357.306,173.710,46.902,159.430
C03372=1032.268,401.093,357.351,173.700,46.898,159.427
C03373=1032.258,400.847,357.396,173.690,46.895,159.425
C03374=1032.248,400.601,357.440,173.680,46.891,159.423
C03375=1032.239,400.355,357.485,173.670,46.887,159.420
C03376=1032.229,400.110,357.530,173.661,46.883,159.418
C03377=1032.219,399.864,357.573,173.651,46.879,159.416
C03378=1032.209,399.619,357.618,173.641,46.876,159.414
C03379=1032.200,399.372,357.662,173.631,46.872,159.412
C03380=1032.190,399.127,357.707,173.621,46.868,159.409
C03381=1032.181,398.881,357.751,173.611,46.865,159.407
C03382=1032.170,398.635,357.796,173.601,46.861,159.405
C03383=1032.160,398.389,357.840,173.592,46.857,159.403
C03384=1032.150,398.143,357.885,173.582,46.853,159.401
C03385=1032.140,397.897,357.928,173.572,46.849,159.398
C03386=1032.131,397.651,357.972,173.562,46.846,159.396
C03387=1032.122,397.406,358.016,173.552,46.842,159.394
C03388=1032.112,397.161,358.060,173.543,46.839,159.392
C03389=1032.102,396.914,358.104,173.533,46.835,159.390
C03390=1032.093,396.668,358.149,173.523,46.831,159.388
C03391=1032.083,396.422,358.193,173.515,46.828,159.385
C03392=1032.073,396.176,358.236,173.505,46.824,159.383
C03393=1032.064,395.930,358.280,173.495,46.821,159.381
C03394=1032.055,395.685,358.324,173.486,46.817,159.379
C03395=1032.045,395.439,358.368,173.476,46.814,159.377
C03396=1032.036,395.193,358.412,173.466,46.810,159.375
C03397=1032.026,394.947,358.456,173.458,46.807,159.373
C03398=1032.017,394.709,358.498,173.448,46.803,159.371
C03399=1032.008,394.471,358.540,173.439,46.800,159.369
C03400=1031.998,394.233,358.582,173.430,46.796,159.367
C03401=1031.990,393.995,358.625,173.421,46.793,159.365
C03402=1031.980,393.756,358.666,173.412,46.790,159.363
C03403=1031.971,393.519,358.709,173.402,46.786,159.361
C03404=1031.962,393.281,358.750,173.394,46.783,159.359
C03405=1031.953,393.043,358.792,173.385,46.780,159.357
C03406=1031.944,392.797,358.836,173.375,46.776,159.355
C03407=1031.934,392.551,358.879,173.367,46.773,159.353
C03408=1031.925,392.305,358.922,173.357,46.770,159.351
C03409=1031.915,392.059,358.966,173.348,46.766,159.349
C03410=1031.906,391.813,359.009,173.338,46.763,159.347
C03411=1031.897,391.566,359.052,173.330,46.760,159.345
C03412=1031.888,391.321,359.095,173.320,46.757,159.343
C03413=1031.878,391.075,359.138,173.312,46.754,159.341
C03414=1031.869,390.828,359.181,173.303,46.750,159.339
C03415=1031.859,390.583,359.225,173.293,46.747,159.337
C03416=1031.851,390.337,359.268,173.285,46.743,159.335
C03417=1031.842,390.091,359.310,173.275,46.741,159.333
C03418=1031.832,389.844,359.353,173.266,46.737,159.331
C03419=1031.823,389.598,359.396,173.258,46.734,159.329
C03420=1031.813,389.352,359.439,173.248,46.731,159.327
C03421=1031.804,389.106,359.481,173.240,46.728,159.325
C03422=1031.796,388.860,359.524,173.231,46.724,159.324
C03423=1031.786,388.614,359.567,173.222,46.722,159.322
C03424=1031.777,388.368,359.609,173.213,46.718,159.320
C03425=1031.768,388.122,359.652,173.205,46.715,159.318
C03426=1031.758,387.875,359.695,173.195,46.712,159.316
C03427=1031.749,387.630,359.738,173.187,46.709,159.314
C03428=1031.741,387.383,359.780,173.178,46.706,159.312
C03429=1031.732,387.137,359.822,173.170,46.703,159.310
C03430=1031.722,386.891,359.865,173.160,46.700,159.309
C03431=1031.712,386.645,359.908,173.152,46.697,159.307
C03432=1031.704,386.399,359.949,173.143,46.694,159.305
C03433=1031.694,386.153,359.992,173.135,46.691,159.303
C03434=1031.685,385.906,360.034,173.126,46.688,159.301
C03435=1031.676,385.660,360.077,173.117,46.685,159.299
C03436=1031.667,385.414,360.119,173.109,46.682,159.298
C03437=1031.658,385.168,360.161,173.100,46.679,159.296
C03438=1031.649,384.921,360.203,173.092,46.676,159.294
C03439=1031.640,384.675,360.245,173.083,46.673,159.292
C03440=1031.631,384.429,360.287,173.074,46.671,159.291
C03441=1031.622,384.183,360.329,173.066,46.668,159.289
C03442=1031.612,383.936,360.371,173.058,46.665,159.287
C03443=1031.604,383.689,360.412,173.049,46.662,159.285
C03444=1031.594,383.444,360.455,173.041,46.659,159.283
C03445=1031.585,383.197,360.497,173.033,46.657,159.282
C03446=1031.576,382.951,360.538,173.024,46.653,159.280
C03447=1031.568,382.705,360.580,173.016,46.651,159.278
C03448=1031.559,382.459,360.621,173.007,46.648,159.276
C03449=1031.550,382.213,360.663,172.999,46.646,159.275
C03450=1031.541,381.966,360.705,172.990,46.642,159.273
C03451=1031.532,381.720,360.747,172.982,46.640,159.271
C03452=1031.523,381.474,360.788,172.974,46.637,159.270
C03453=1031.515,381.227,360.830,172.966,46.634,159.268
C03454=1031.506,380.981,360.872,172.957,46.632,159.266
C03455=1031.497,380.734,360.913,172.949,46.629,159.265
C03456=1031.488,380.488,360.956,172.941,46.627,159.263
C03457=1031.480,380.242,360.997,172.933,46.624,159.261
C03458=1031.472,380.022,361.034,172.926,46.621,159.260
C03459=1031.464,379.801,361.071,172.919,46.619,159.258
C03460=1031.456,379.581,361.108,172.911,46.617,159.257
C03461=1031.448,379.360,361.145,172.904,46.614,159.255
C03462=1031.441,379.140,361.182,172.897,46.612,159.254
C03463=1031.433,378.920,361.220,172.890,46.609,159.252
C03464=1031.425,378.699,361.256,172.882,46.607,159.251
C03465=1031.418,378.479,361.294,172.875,46.605,159.249
C03466=1031.409,378.232,361.335,172.867,46.602,159.248
C03467=1031.401,377.986,361.376,172.859,46.599,159.246
C03468=1031.392,377.739,361.417,172.851,46.597,159.245
C03469=1031.383,377.493,361.459,172.844,46.595,159.243
C03470=1031.374,377.247,361.499,172.836,46.592,159.241
C03471=1031.366,377.001,361.540,172.828,46.590,159.240
C03472=1031.357,376.754,361.581,172.820,46.587,159.238
C03473=1031.349,376.507,361.622,172.812,46.585,159.237
C03474=1031.340,376.261,361.662,172.804,46.582,159.235
C03475=1031.331,376.014,361.704,172.795,46.580,159.234
C03476=1031.323,375.768,361.745,172.788,46.577,159.232
C03477=1031.313,375.521,361.785,172.781,46.575,159.231
C03478=1031.305,375.275,361.826,172.772,46.573,159.229
C03479=1031.297,375.028,361.867,172.765,46.571,159.227
C03480=1031.288,374.782,361.907,172.756,46.568,159.226
C03481=1031.279,374.536,361.949,172.750,46.566,159.224
C03482=1031.271,374.289,361.989,172.741,46.563,159.223
C03483=1031.261,374.043,362.030,172.733,46.561,159.221
C03484=1031.253,373.797,362.070,172.726,46.559,159.220
C03485=1031.245,373.550,362.111,172.719,46.556,159.218
C03486=1031.236,373.303,362.151,172.711,46.554,159.217
C03487=1031.228,373.056,362.192,172.703,46.552,159.215
C03488=1031.220,372.810,362.232,172.696,46.549,159.214
C03489=1031.211,372.564,362.272,172.688,46.547,159.212
C03490=1031.202,372.317,362.313,172.680,46.545,159.211
C03491=1031.194,372.070,362.354,172.673,46.542,159.209
C03492=1031.186,371.824,362.394,172.665,46.540,159.208
C03493=1031.177,371.577,362.434,172.657,46.538,159.206
C03494=1031.169,371.331,362.475,172.650,46.536,159.205
C03495=1031.160,371.085,362.515,172.642,46.533,159.203
C03496=1031.152,370.837,362.555,172.635,46.531,159.202
C03497=1031.144,370.591,362.596,172.628,46.529,159.201
C03498=1031.135,370.345,362.636,172.620,46.527,159.199
C03499=1031.128,370.098,362.676,172.612,46.525,159.198
C03500=1031.120,369.852,362.716,172.605,46.523,159.196
C03501=1031.110,369.604,362.756,172.597,46.521,159.195
C03502=1031.102,369.358,362.797,172.591,46.519,159.193
C03503=1031.094,369.111,362.836,172.583,46.517,159.192
C03504=1031.086,368.865,362.877,172.576,46.514,159.191
C03505=1031.077,368.618,362.916,172.568,46.512,159.189
C03506=1031.068,368.371,362.956,172.560,46.510,159.188
C03507=1031.061,368.124,362.996,172.554,46.508,159.186
C03508=1031.052,367.878,363.036,172.546,46.506,159.185
C03509=1031.044,367.632,363.075,172.539,46.504,159.184
C03510=1031.036,367.385,363.115,172.531,46.502,159.182
C03511=1031.027,367.138,363.155,172.525,46.500,159.181
C03512=1031.018,366.891,363.194,172.517,46.498,159.180
C03513=1031.011,366.644,363.234,172.510,46.496,159.178
C03514=1031.002,366.398,363.274,172.502,46.494,159.177
C03515=1030.993,366.151,363.313,172.496,46.492,159.176
C03516=1030.986,365.905,363.353,172.488,46.491,159.174
C03517=1030.977,365.658,363.392,172.481,46.488,159.173
C03518=1030.970,365.448,363.426,172.475,46.487,159.172
C03519=1030.963,365.238,363.460,172.468,46.485,159.171
C03520=1030.956,365.028,363.493,172.463,46.484,159.170
C03521=1030.950,364.817,363.527,172.457,46.482,159.168
C03522=1030.942,364.608,363.561,172.451,46.480,159.167
C03523=1030.936,364.398,363.594,172.445,46.478,159.166
C03524=1030.929,364.189,363.628,172.438,46.477,159.165
C03525=1030.922,363.978,363.661,172.433,46.475,159.164
C03526=1030.913,363.732,363.700,172.425,46.474,159.163
C03527=1030.906,363.485,363.740,172.419,46.472,159.161
C03528=1030.897,363.238,363.779,172.411,46.470,159.160
C03529=1030.889,362.991,363.818,172.404,46.468,159.159
C03530=1030.881,362.744,363.858,172.398,46.466,159.157
C03531=1030.873,362.498,363.897,172.390,46.465,159.156
C03532=1030.865,362.251,363.935,172.383,46.463,159.155
C03533=1030.857,362.004,363.975,172.377,46.461,159.154
C03534=1030.849,361.757,364.014,172.369,46.459,159.152
C03535=1030.841,361.510,364.053,172.363,46.457,159.151
C03536=1030.833,361.264,364.092,172.356,46.455,159.150
C03537=1030.826,361.017,364.131,172.349,46.454,159.149
C03538=1030.817,360.770,364.171,172.342,46.452,159.147
C03539=1030.809,360.523,364.209,172.336,46.451,159.146
C03540=1030.801,360.276,364.248,172.328,46.449,159.145
C03541=1030.793,360.030,364.287,172.321,46.447,159.144
C03542=1030.785,359.783,364.326,172.315,46.445,159.142
C03543=1030.777,359.536,364.364,172.307,46.444,159.141
C03544=1030.768,359.289,364.403,172.301,46.442,159.140
C03545=1030.761,359.042,364.442,172.294,46.440,159.139
C03546=1030.753,358.795,364.480,172.288,46.439,159.138
C03547=1030.744,358.548,364.519,172.280,46.437,159.136
C03548=1030.737,358.302,364.558,172.274,46.435,159.135
C03549=1030.728,358.055,364.597,172.267,46.434,159.134
C03550=1030.720,357.808,364.635,172.261,46.433,159.133
C03551=1030.713,357.561,364.673,172.253,46.431,159.132
C03552=1030.705,357.314,364.712,172.247,46.429,159.130
C03553=1030.696,357.067,364.751,172.240,46.428,159.129
C03554=1030.689,356.820,364.789,172.234,46.426,159.128
C03555=1030.681,356.573,364.827,172.227,46.425,159.127
C03556=1030.673,356.326,364.866,172.220,46.423,159.126
C03557=1030.665,356.079,364.904,172.214,46.422,159.125
C03558=1030.657,355.832,364.943,172.207,46.420,159.123
C03559=1030.649,355.586,364.981,172.201,46.419,159.122
C03560=1030.641,355.338,365.020,172.193,46.417,159.121
C03561=1030.634,355.092,365.058,172.187,46.416,159.120
C03562=1030.625,354.844,365.095,172.181,46.415,159.119
C03563=1030.618,354.598,365.134,172.174,46.413,159.118
C03564=1030.609,354.351,365.172,172.168,46.411,159.117
C03565=1030.602,354.104,365.210,172.162,46.410,159.116
C03566=1030.594,353.856,365.248,172.154,46.409,159.114
C03567=1030.586,353.610,365.286,172.148,46.408,159.113
C03568=1030.578,353.363,365.325,172.141,46.406,159.112
C03569=1030.570,353.116,365.362,172.135,46.405,159.111
C03570=1030.563,352.869,365.400,172.129,46.403,159.110
C03571=1030.554,352.622,365.438,172.122,46.402,159.109
C03572=1030.547,352.375,365.476,172.116,46.401,159.108
C03573=1030.538,352.128,365.514,172.110,46.399,159.107
C03574=1030.531,351.881,365.552,172.103,46.398,159.106
C03575=1030.523,351.635,365.590,172.096,46.396,159.105
C03576=1030.515,351.387,365.628,172.090,46.395,159.104
C03577=1030.508,351.140,365.666,172.084,46.394,159.103
C03578=1030.495,350.726,365.729,172.073,46.391,159.101
C03579=1030.481,350.313,365.792,172.062,46.389,159.099
C03580=1030.469,349.899,365.855,172.052,46.387,159.097
C03581=1030.456,349.486,365.918,172.041,46.385,159.095
C03582=1030.448,349.239,365.956,172.035,46.384,159.094
C03583=1030.441,348.992,365.993,172.028,46.383,159.093
C03584=1030.432,348.744,366.031,172.022,46.382,159.092
C03585=1030.425,348.497,366.068,172.016,46.381,159.091
C03586=1030.418,348.250,366.106,172.010,46.379,159.090
C03587=1030.410,348.003,366.143,172.003,46.378,159.089
C03588=1030.402,347.756,366.181,171.997,46.377,159.088
C03589=1030.394,347.509,366.218,171.991,46.376,159.087
C03590=1030.387,347.262,366.256,171.985,46.375,159.086
C03591=1030.379,347.015,366.293,171.979,46.373,159.085
C03592=1030.371,346.768,366.330,171.972,46.372,159.084
C03593=1030.363,346.521,366.367,171.966,46.372,159.083
C03594=1030.356,346.273,366.404,171.960,46.371,159.082
C03595=1030.348,346.026,366.441,171.954,46.370,159.081
C03596=1030.341,345.779,366.479,171.948,46.368,159.080
C03597=1030.333,345.532,366.516,171.942,46.367,159.079
C03598=1030.325,345.285,366.553,171.936,46.366,159.078
C03599=1030.317,345.038,366.590,171.930,46.365,159.077
C03600=1030.310,344.791,366.628,171.924,46.364,159.076
C03601=1030.302,344.544,366.664,171.918,46.363,159.075
C03602=1030.295,344.297,366.702,171.912,46.362,159.074
C03603=1030.287,344.050,366.738,171.906,46.361,159.073
C03604=1030.280,343.803,366.776,171.899,46.360,159.072
C03605=1030.272,343.555,366.812,171.894,46.359,159.072
C03606=1030.264,343.308,366.849,171.887,46.358,159.071
C03607=1030.257,343.061,366.887,171.881,46.357,159.070
C03608=1030.249,342.814,366.923,171.875,46.356,159.069
C03609=1030.242,342.567,366.960,171.869,46.355,159.068
C03610=1030.234,342.319,366.997,171.864,46.354,159.067
C03611=1030.226,342.072,367.034,171.858,46.353,159.066
C03612=1030.219,341.825,367.071,171.852,46.352,159.065
C03613=1030.212,341.578,367.107,171.846,46.351,159.064
C03614=1030.204,341.331,367.145,171.840,46.350,159.063
C03615=1030.197,341.083,367.181,171.833,46.349,159.062
C03616=1030.189,340.836,367.217,171.828,46.349,159.061
C03617=1030.182,340.589,367.254,171.822,46.347,159.060
C03618=1030.175,340.342,367.291,171.816,46.347,159.060
C03619=1030.167,340.095,367.328,171.810,46.346,159.059
C03620=1030.159,339.848,367.364,171.804,46.345,159.058
C03621=1030.151,339.600,367.400,171.798,46.344,159.057
C03622=1030.144,339.352,367.437,171.792,46.343,159.056
C03623=1030.136,339.106,367.474,171.787,46.343,159.055
C03624=1030.129,338.859,367.510,171.781,46.341,159.054
C03625=1030.122,338.611,367.546,171.775,46.341,159.053
C03626=1030.114,338.364,367.582,171.769,46.340,159.053
C03627=1030.106,338.116,367.618,171.763,46.339,159.052
C03628=1030.099,337.869,367.654,171.758,46.338,159.051
C03629=1030.092,337.623,367.692,171.752,46.338,159.050
C03630=1030.084,337.375,367.728,171.746,46.337,159.049
C03631=1030.077,337.128,367.764,171.740,46.336,159.048
C03632=1030.069,336.880,367.800,171.734,46.336,159.047
C03633=1030.062,336.633,367.836,171.729,46.335,159.047
C03634=1030.049,336.216,367.898,171.720,46.334,159.045
C03635=1030.037,335.800,367.958,171.710,46.332,159.044
C03636=1030.024,335.383,368.019,171.701,46.331,159.042
